KUKA KRL program: EPS_2_251806_MH58A_A_20260212042255.src

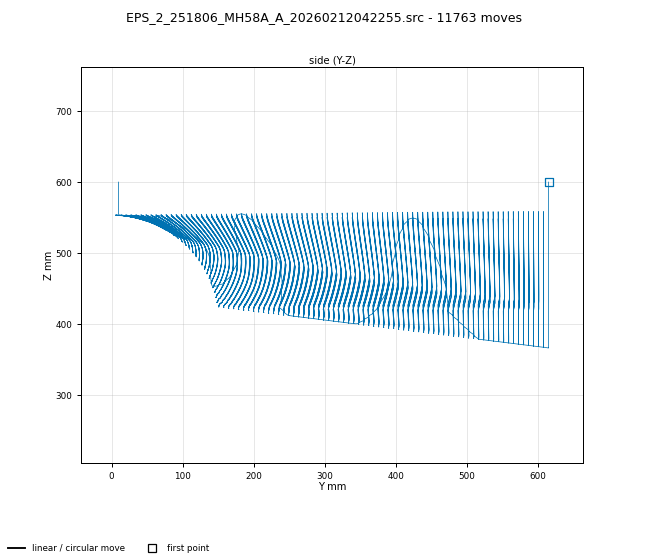
[picture p0: tool path of EPS_2_251806_MH58A_A_20260212042255.src, 11763 of 11765 moves have a stored position in this frame; points joined in program order, loops and branches not executed]
&ACCESS RVP
&REL 4
&COMMENT QRS 19112012
&PARAM EDITMASK = *
DEF PART()
EXT BAS (BAS_COMMAND :IN,REAL :IN )
INT I
BAS (#INITMOV,0 )

;KUKA QRS Post kuka4.cps  Date:22-06-2017 !

File_ID=3025

QRS_PRE_INIT()

;Init var - Until changes are made in qrs_pre_init
Outlet_Square_prg=0
Inlet_1_Square_prg=0
Inlet_2_Square_prg=0
Inlet_3_Square_prg=0
Inlet_4_Square_prg=0
Inlet_5_Square_prg=0

Outlet_1={X 0.000, Y 515.060, Z 433.000, B 0.000, E1 0.000 }
Inlet_1={X 0.000, Y 515.800, Z 423.000, B 0.000, E1 180.000 }
Outlet_1_type=251
Inlet_1_type=251
;QRS#1=Sidecore dimensions
;QRS#2=250-10" PVC SDR 35
;QRS#3=250-10" PVC SDR 35
;QRS#4=
;QRS#5=
;QRS#6=
;QRS#7=
;QRS#8=
;QRS#9=14M PSX
;QRS#10=14M PSX
;QRS#11=
;QRS#12=
;QRS#13=
;QRS#14=
;QRS#15=
;QRS#16=1220x127x838 2,75'
;QRS#17=EPS Height
;QRS#18=558,5
;QRS#19=*
;QRS#20= UPDATED VERSION 22-06-2017
;QRS#21=*
Outlet_Square=0100
Inlet_1_Square=0100
Inlet_2_Square=0
Inlet_3_Square=0
Inlet_4_Square=0
Inlet_5_Square=0
Mill_Square=1
Outlet_Square_Prg=205
Inlet_1_Square_prg=205

QRS_INIT()

$ADVANCE=5

; T1
PTP {E1 173.605,E2 173.605}
PTP {X 0,Y 615.509,A -85,B 0,C 180,E1 173.605,E2 173.605,E3 0,E4 0,E5 0,E6 0}
QRS_SPEED_INIT()
LIN {X 0,Y 615.509,Z 600,A -85,B 0,C 180,E1 173.605,E2 173.605,E3 0,E4 0,E5 0,E6 0} C_VEL
LIN {X 0,Y 615.509,Z 376.499,A -85,B 0,C 180,E1 173.605,E2 173.605} C_VEL
LIN {X 0,Y 615.509,Z 368.324,A -85,B 0,C 180,E1 173.605,E2 173.605} C_VEL
LIN {X 0,Y 615.493,Z 366.324,A -85,B 0,C 180,E1 173.419,E2 173.419} C_VEL
LIN {X 0,Y 615.489,Z 366.315,A -85,B 0,C 180,E1 170.801,E2 170.801} C_VEL
LIN {X 0,Y 615.48,Z 366.318,A -85,B 0,C 180,E1 168.139,E2 168.139} C_VEL
LIN {X 0,Y 615.484,Z 366.327,A -85,B 0,C 180,E1 165.451,E2 165.451} C_VEL
LIN {X 0,Y 615.495,Z 366.313,A -85,B 0,C 180,E1 162.73,E2 162.73} C_VEL
LIN {X 0,Y 615.49,Z 366.315,A -85,B 0,C 180,E1 159.967,E2 159.967} C_VEL
LIN {X 0,Y 615.497,Z 366.322,A -85,B 0,C 180,E1 157.156,E2 157.156} C_VEL
LIN {X 0,Y 615.481,Z 366.322,A -85,B 0,C 180,E1 154.284,E2 154.284} C_VEL
LIN {X 0,Y 615.478,Z 366.316,A -85,B 0,C 180,E1 151.552,E2 151.552} C_VEL
LIN {X 0,Y 615.487,Z 366.321,A -85,B 0,C 180,E1 148.914,E2 148.914} C_VEL
LIN {X 0,Y 615.478,Z 366.318,A -85,B 0,C 180,E1 146.467,E2 146.467} C_VEL
LIN {X 0,Y 615.497,Z 366.322,A -85,B 0,C 180,E1 144.165,E2 144.165} C_VEL
LIN {X 0,Y 615.483,Z 366.315,A -85,B 0,C 180,E1 141.931,E2 141.931} C_VEL
LIN {X 0,Y 615.49,Z 366.326,A -85,B 0,C 180,E1 139.394,E2 139.394} C_VEL
LIN {X 0,Y 615.478,Z 366.317,A -85,B 0,C 180,E1 136.754,E2 136.754} C_VEL
LIN {X 0,Y 615.481,Z 366.317,A -85,B 0,C 180,E1 133.997,E2 133.997} C_VEL
LIN {X 0,Y 615.488,Z 366.323,A -85,B 0,C 180,E1 131.474,E2 131.474} C_VEL
LIN {X 0,Y 615.478,Z 366.316,A -85,B 0,C 180,E1 128.905,E2 128.905} C_VEL
LIN {X 0,Y 615.486,Z 366.82,A -85,B 0,C 180,E1 128.011,E2 128.011} C_VEL
LIN {X 0,Y 615.487,Z 371.423,A -85,B 0,C 180,E1 125.616,E2 125.616} C_VEL
LIN {X 0,Y 615.485,Z 376.105,A -85,B 0,C 180,E1 123.236,E2 123.236} C_VEL
LIN {X 0,Y 615.478,Z 380.808,A -85,B 0,C 180,E1 120.92,E2 120.92} C_VEL
LIN {X 0,Y 615.491,Z 385.941,A -85,B 0,C 180,E1 118.45,E2 118.45} C_VEL
LIN {X 0,Y 615.498,Z 392.089,A -85,B 0,C 180,E1 115.57,E2 115.57} C_VEL
LIN {X 0,Y 615.492,Z 398.04,A -85,B 0,C 180,E1 112.844,E2 112.844} C_VEL
LIN {X 0,Y 615.479,Z 404.312,A -85,B 0,C 180,E1 110.033,E2 110.033} C_VEL
LIN {X 0,Y 615.481,Z 410.569,A -85,B 0,C 180,E1 107.271,E2 107.271} C_VEL
LIN {X 0,Y 615.481,Z 416.835,A -85,B 0,C 180,E1 104.549,E2 104.549} C_VEL
LIN {X 0,Y 615.483,Z 418.133,A -85,B 0,C 180,E1 103.989,E2 103.989} C_VEL
LIN {X 0,Y 615.486,Z 434.986,A -85,B 0,C 180,E1 103.664,E2 103.664} C_VEL
LIN {X 0,Y 615.478,Z 449.325,A -85,B 0,C 180,E1 103.243,E2 103.243} C_VEL
LIN {X 0,Y 615.487,Z 462.901,A -85,B 0,C 180,E1 102.698,E2 102.698} C_VEL
LIN {X 0,Y 615.486,Z 475.843,A -85,B 0,C 180,E1 102.028,E2 102.028} C_VEL
LIN {X 0,Y 615.499,Z 487.559,A -85,B 0,C 180,E1 101.276,E2 101.276} C_VEL
LIN {X 0,Y 615.498,Z 499.226,A -85,B 0,C 180,E1 100.36,E2 100.36} C_VEL
LIN {X 0,Y 615.497,Z 509.65,A -85,B 0,C 180,E1 99.364,E2 99.364} C_VEL
LIN {X 0,Y 615.496,Z 518.24,A -85,B 0,C 180,E1 98.371,E2 98.371} C_VEL
LIN {X 0,Y 615.495,Z 526.453,A -85,B 0,C 180,E1 97.216,E2 97.216} C_VEL
LIN {X 0,Y 615.496,Z 532.184,A -85,B 0,C 180,E1 96.227,E2 96.227} C_VEL
LIN {X 0,Y 615.494,Z 536.887,A -85,B 0,C 180,E1 95.241,E2 95.241} C_VEL
LIN {X 0,Y 615.496,Z 541.757,A -85,B 0,C 180,E1 93.928,E2 93.928} C_VEL
LIN {X 0,Y 615.496,Z 545.154,A -85,B 0,C 180,E1 92.618,E2 92.618} C_VEL
LIN {X 0,Y 615.493,Z 547.174,A -85,B 0,C 180,E1 91.309,E2 91.309} C_VEL
LIN {X 0,Y 615.494,Z 547.884,A -85,B 0,C 180,E1 90,E2 90} C_VEL
LIN {X 0,Y 615.49,Z 547.28,A -85,B 0,C 180,E1 88.691,E2 88.691} C_VEL
LIN {X 0,Y 615.493,Z 545.35,A -85,B 0,C 180,E1 87.382,E2 87.382} C_VEL
LIN {X 0,Y 615.496,Z 542.045,A -85,B 0,C 180,E1 86.071,E2 86.071} C_VEL
LIN {X 0,Y 615.496,Z 537.273,A -85,B 0,C 180,E1 84.759,E2 84.759} C_VEL
LIN {X 0,Y 615.495,Z 530.874,A -85,B 0,C 180,E1 83.443,E2 83.443} C_VEL
LIN {X 0,Y 615.496,Z 523.743,A -85,B 0,C 180,E1 82.289,E2 82.289} C_VEL
LIN {X 0,Y 615.497,Z 516.27,A -85,B 0,C 180,E1 81.298,E2 81.298} C_VEL
LIN {X 0,Y 615.496,Z 507.29,A -85,B 0,C 180,E1 80.304,E2 80.304} C_VEL
LIN {X 0,Y 615.499,Z 496.204,A -85,B 0,C 180,E1 79.291,E2 79.291} C_VEL
LIN {X 0,Y 615.498,Z 485.279,A -85,B 0,C 180,E1 78.473,E2 78.473} C_VEL
LIN {X 0,Y 615.479,Z 472.982,A -85,B 0,C 180,E1 77.721,E2 77.721} C_VEL
LIN {X 0,Y 615.488,Z 461.143,A -85,B 0,C 180,E1 77.134,E2 77.134} C_VEL
LIN {X 0,Y 615.476,Z 448.216,A -85,B 0,C 180,E1 76.63,E2 76.63} C_VEL
LIN {X 0,Y 615.492,Z 435.233,A -85,B 0,C 180,E1 76.252,E2 76.252} C_VEL
LIN {X 0,Y 615.482,Z 420.854,A -85,B 0,C 180,E1 75.971,E2 75.971} C_VEL
LIN {X 0,Y 615.48,Z 418.118,A -85,B 0,C 180,E1 75.914,E2 75.914} C_VEL
LIN {X 0,Y 615.489,Z 412.342,A -85,B 0,C 180,E1 73.413,E2 73.413} C_VEL
LIN {X 0,Y 615.484,Z 406.076,A -85,B 0,C 180,E1 70.662,E2 70.662} C_VEL
LIN {X 0,Y 615.478,Z 399.81,A -85,B 0,C 180,E1 67.863,E2 67.863} C_VEL
LIN {X 0,Y 615.492,Z 393.538,A -85,B 0,C 180,E1 65.008,E2 65.008} C_VEL
LIN {X 0,Y 615.484,Z 388.839,A -85,B 0,C 180,E1 62.823,E2 62.823} C_VEL
LIN {X 0,Y 615.482,Z 383.318,A -85,B 0,C 180,E1 60.207,E2 60.207} C_VEL
LIN {X 0,Y 615.489,Z 377.849,A -85,B 0,C 180,E1 57.542,E2 57.542} C_VEL
LIN {X 0,Y 615.483,Z 373.159,A -85,B 0,C 180,E1 55.184,E2 55.184} C_VEL
LIN {X 0,Y 615.488,Z 368.46,A -85,B 0,C 180,E1 52.758,E2 52.758} C_VEL
LIN {X 0,Y 615.494,Z 366.881,A -85,B 0,C 180,E1 51.932,E2 51.932} C_VEL
LIN {X 0,Y 615.482,Z 366.315,A -85,B 0,C 180,E1 50.939,E2 50.939} C_VEL
LIN {X 0,Y 615.493,Z 366.325,A -85,B 0,C 180,E1 48.526,E2 48.526} C_VEL
LIN {X 0,Y 615.491,Z 366.315,A -85,B 0,C 180,E1 45.85,E2 45.85} C_VEL
LIN {X 0,Y 615.483,Z 366.315,A -85,B 0,C 180,E1 43.047,E2 43.047} C_VEL
LIN {X 0,Y 615.495,Z 366.322,A -85,B 0,C 180,E1 40.606,E2 40.606} C_VEL
LIN {X 0,Y 615.483,Z 366.315,A -85,B 0,C 180,E1 38.011,E2 38.011} C_VEL
LIN {X 0,Y 615.498,Z 366.325,A -85,B 0,C 180,E1 35.615,E2 35.615} C_VEL
LIN {X 0,Y 615.482,Z 366.315,A -85,B 0,C 180,E1 33.237,E2 33.237} C_VEL
LIN {X 0,Y 615.494,Z 366.322,A -85,B 0,C 180,E1 30.919,E2 30.919} C_VEL
LIN {X 0,Y 615.478,Z 366.316,A -85,B 0,C 180,E1 28.448,E2 28.448} C_VEL
LIN {X 0,Y 615.489,Z 366.322,A -85,B 0,C 180,E1 25.716,E2 25.716} C_VEL
LIN {X 0,Y 615.495,Z 366.321,A -85,B 0,C 180,E1 22.844,E2 22.844} C_VEL
LIN {X 0,Y 615.491,Z 366.314,A -85,B 0,C 180,E1 20.033,E2 20.033} C_VEL
LIN {X 0,Y 615.494,Z 366.314,A -85,B 0,C 180,E1 17.27,E2 17.27} C_VEL
LIN {X 0,Y 615.489,Z 366.327,A -85,B 0,C 180,E1 14.549,E2 14.549} C_VEL
LIN {X 0,Y 615.477,Z 366.318,A -85,B 0,C 180,E1 11.861,E2 11.861} C_VEL
LIN {X 0,Y 615.489,Z 366.316,A -85,B 0,C 180,E1 9.199,E2 9.199} C_VEL
LIN {X 0,Y 615.492,Z 366.324,A -85,B 0,C 180,E1 6.557,E2 6.557} C_VEL
LIN {X 0,Y 615.478,Z 366.316,A -85,B 0,C 180,E1 3.929,E2 3.929} C_VEL
LIN {X 0,Y 615.487,Z 366.32,A -85,B 0,C 180,E1 1.309,E2 1.309} C_VEL
LIN {X 0,Y 615.487,Z 366.319,A -85,B 0,C 180,E1 -1.309,E2 -1.309} C_VEL
LIN {X 0,Y 615.477,Z 366.317,A -85,B 0,C 180,E1 -3.929,E2 -3.929} C_VEL
LIN {X 0,Y 615.493,Z 366.325,A -85,B 0,C 180,E1 -6.58,E2 -6.58} C_VEL
LIN {X 0,Y 615.489,Z 366.315,A -85,B 0,C 180,E1 -9.199,E2 -9.199} C_VEL
LIN {X 0,Y 615.48,Z 366.318,A -85,B 0,C 180,E1 -11.861,E2 -11.861} C_VEL
LIN {X 0,Y 615.491,Z 366.325,A -85,B 0,C 180,E1 -14.549,E2 -14.549} C_VEL
LIN {X 0,Y 615.492,Z 366.314,A -85,B 0,C 180,E1 -17.27,E2 -17.27} C_VEL
LIN {X 0,Y 615.493,Z 366.314,A -85,B 0,C 180,E1 -20.033,E2 -20.033} C_VEL
LIN {X 0,Y 615.495,Z 366.322,A -85,B 0,C 180,E1 -22.844,E2 -22.844} C_VEL
LIN {X 0,Y 615.478,Z 366.323,A -85,B 0,C 180,E1 -25.716,E2 -25.716} C_VEL
LIN {X 0,Y 615.478,Z 366.316,A -85,B 0,C 180,E1 -28.448,E2 -28.448} C_VEL
LIN {X 0,Y 615.486,Z 366.321,A -85,B 0,C 180,E1 -31.085,E2 -31.085} C_VEL
LIN {X 0,Y 615.478,Z 366.318,A -85,B 0,C 180,E1 -33.532,E2 -33.532} C_VEL
LIN {X 0,Y 615.496,Z 366.322,A -85,B 0,C 180,E1 -35.834,E2 -35.834} C_VEL
LIN {X 0,Y 615.483,Z 366.315,A -85,B 0,C 180,E1 -38.069,E2 -38.069} C_VEL
LIN {X 0,Y 615.494,Z 366.325,A -85,B 0,C 180,E1 -40.606,E2 -40.606} C_VEL
LIN {X 0,Y 615.478,Z 366.318,A -85,B 0,C 180,E1 -43.246,E2 -43.246} C_VEL
LIN {X 0,Y 615.482,Z 366.316,A -85,B 0,C 180,E1 -46.003,E2 -46.003} C_VEL
LIN {X 0,Y 615.488,Z 366.324,A -85,B 0,C 180,E1 -48.526,E2 -48.526} C_VEL
LIN {X 0,Y 615.478,Z 366.316,A -85,B 0,C 180,E1 -51.095,E2 -51.095} C_VEL
LIN {X 0,Y 615.492,Z 366.45,A -85,B 0,C 180,E1 -51.724,E2 -51.724} C_VEL
LIN {X 0,Y 615.487,Z 372.465,A -85,B 0,C 180,E1 -54.384,E2 -54.384} C_VEL
LIN {X 0,Y 615.485,Z 378.035,A -85,B 0,C 180,E1 -56.763,E2 -56.763} C_VEL
LIN {X 0,Y 615.478,Z 383.591,A -85,B 0,C 180,E1 -59.08,E2 -59.08} C_VEL
LIN {X 0,Y 615.491,Z 389.648,A -85,B 0,C 180,E1 -61.549,E2 -61.549} C_VEL
LIN {X 0,Y 615.498,Z 396.905,A -85,B 0,C 180,E1 -64.429,E2 -64.429} C_VEL
LIN {X 0,Y 615.493,Z 403.92,A -85,B 0,C 180,E1 -67.156,E2 -67.156} C_VEL
LIN {X 0,Y 615.479,Z 411.32,A -85,B 0,C 180,E1 -69.967,E2 -69.967} C_VEL
LIN {X 0,Y 615.487,Z 418.695,A -85,B 0,C 180,E1 -72.729,E2 -72.729} C_VEL
LIN {X 0,Y 615.483,Z 426.086,A -85,B 0,C 180,E1 -75.451,E2 -75.451} C_VEL
LIN {X 0,Y 615.485,Z 427.541,A -85,B 0,C 180,E1 -75.97,E2 -75.97} C_VEL
LIN {X 0,Y 615.494,Z 441.452,A -85,B 0,C 180,E1 -76.21,E2 -76.21} C_VEL
LIN {X 0,Y 615.479,Z 455.537,A -85,B 0,C 180,E1 -76.588,E2 -76.588} C_VEL
LIN {X 0,Y 615.488,Z 468.121,A -85,B 0,C 180,E1 -77.051,E2 -77.051} C_VEL
LIN {X 0,Y 615.484,Z 480.577,A -85,B 0,C 180,E1 -77.637,E2 -77.637} C_VEL
LIN {X 0,Y 615.498,Z 493.318,A -85,B 0,C 180,E1 -78.39,E2 -78.39} C_VEL
LIN {X 0,Y 615.498,Z 504.479,A -85,B 0,C 180,E1 -79.199,E2 -79.199} C_VEL
LIN {X 0,Y 615.499,Z 515.176,A -85,B 0,C 180,E1 -80.138,E2 -80.138} C_VEL
LIN {X 0,Y 615.498,Z 524.542,A -85,B 0,C 180,E1 -81.133,E2 -81.133} C_VEL
LIN {X 0,Y 615.494,Z 532.302,A -85,B 0,C 180,E1 -82.124,E2 -82.124} C_VEL
LIN {X 0,Y 615.496,Z 538.651,A -85,B 0,C 180,E1 -83.1,E2 -83.1} C_VEL
LIN {X 0,Y 615.499,Z 544.069,A -85,B 0,C 180,E1 -84.101,E2 -84.101} C_VEL
LIN {X 0,Y 615.495,Z 549.682,A -85,B 0,C 180,E1 -85.415,E2 -85.415} C_VEL
LIN {X 0,Y 615.495,Z 553.754,A -85,B 0,C 180,E1 -86.727,E2 -86.727} C_VEL
LIN {X 0,Y 615.499,Z 556.405,A -85,B 0,C 180,E1 -88.037,E2 -88.037} C_VEL
LIN {X 0,Y 615.494,Z 557.723,A -85,B 0,C 180,E1 -89.346,E2 -89.346} C_VEL
LIN {X 0,Y 615.494,Z 557.723,A -85,B 0,C 180,E1 -90.654,E2 -90.654} C_VEL
LIN {X 0,Y 615.499,Z 556.405,A -85,B 0,C 180,E1 -91.963,E2 -91.963} C_VEL
LIN {X 0,Y 615.495,Z 553.754,A -85,B 0,C 180,E1 -93.273,E2 -93.273} C_VEL
LIN {X 0,Y 615.495,Z 549.683,A -85,B 0,C 180,E1 -94.584,E2 -94.584} C_VEL
LIN {X 0,Y 615.499,Z 544.07,A -85,B 0,C 180,E1 -95.898,E2 -95.898} C_VEL
LIN {X 0,Y 615.496,Z 538.652,A -85,B 0,C 180,E1 -96.9,E2 -96.9} C_VEL
LIN {X 0,Y 615.496,Z 531.073,A -85,B 0,C 180,E1 -98.041,E2 -98.041} C_VEL
LIN {X 0,Y 615.498,Z 521.588,A -85,B 0,C 180,E1 -99.199,E2 -99.199} C_VEL
LIN {X 0,Y 615.498,Z 511.642,A -85,B 0,C 180,E1 -100.194,E2 -100.194} C_VEL
LIN {X 0,Y 615.498,Z 500.384,A -85,B 0,C 180,E1 -101.118,E2 -101.118} C_VEL
LIN {X 0,Y 615.497,Z 489.415,A -85,B 0,C 180,E1 -101.861,E2 -101.861} C_VEL
LIN {X 0,Y 615.486,Z 477.329,A -85,B 0,C 180,E1 -102.53,E2 -102.53} C_VEL
LIN {X 0,Y 615.48,Z 463.93,A -85,B 0,C 180,E1 -103.117,E2 -103.117} C_VEL
LIN {X 0,Y 615.485,Z 449.896,A -85,B 0,C 180,E1 -103.58,E2 -103.58} C_VEL
LIN {X 0,Y 615.493,Z 435.698,A -85,B 0,C 180,E1 -103.904,E2 -103.904} C_VEL
LIN {X 0,Y 615.484,Z 427.449,A -85,B 0,C 180,E1 -104.049,E2 -104.049} C_VEL
LIN {X 0,Y 615.489,Z 420.545,A -85,B 0,C 180,E1 -106.587,E2 -106.587} C_VEL
LIN {X 0,Y 615.487,Z 413.158,A -85,B 0,C 180,E1 -109.338,E2 -109.338} C_VEL
LIN {X 0,Y 615.478,Z 405.775,A -85,B 0,C 180,E1 -112.137,E2 -112.137} C_VEL
LIN {X 0,Y 615.49,Z 398.379,A -85,B 0,C 180,E1 -114.992,E2 -114.992} C_VEL
LIN {X 0,Y 615.481,Z 392.839,A -85,B 0,C 180,E1 -117.177,E2 -117.177} C_VEL
LIN {X 0,Y 615.477,Z 386.338,A -85,B 0,C 180,E1 -119.793,E2 -119.793} C_VEL
LIN {X 0,Y 615.495,Z 379.886,A -85,B 0,C 180,E1 -122.457,E2 -122.457} C_VEL
LIN {X 0,Y 615.484,Z 374.318,A -85,B 0,C 180,E1 -124.815,E2 -124.815} C_VEL
LIN {X 0,Y 615.486,Z 368.759,A -85,B 0,C 180,E1 -127.242,E2 -127.242} C_VEL
LIN {X 0,Y 615.487,Z 366.32,A -85,B 0,C 180,E1 -128.381,E2 -128.381} C_VEL
LIN {X 0,Y 615.484,Z 366.321,A -85,B 0,C 180,E1 -131.094,E2 -131.094} C_VEL
LIN {X 0,Y 615.492,Z 366.319,A -85,B 0,C 180,E1 -133.244,E2 -133.244} C_VEL
LIN {X 0,Y 615.483,Z 366.323,A -85,B 0,C 180,E1 -136.003,E2 -136.003} C_VEL
LIN {X 0,Y 615.482,Z 366.317,A -85,B 0,C 180,E1 -138.906,E2 -138.906} C_VEL
LIN {X 0,Y 615.495,Z 366.326,A -85,B 0,C 180,E1 -141.096,E2 -141.096} C_VEL
LIN {X 0,Y 615.478,Z 366.316,A -85,B 0,C 180,E1 -143.575,E2 -143.575} C_VEL
LIN {X 0,Y 615.495,Z 366.325,A -85,B 0,C 180,E1 -145.978,E2 -145.978} C_VEL
LIN {X 0,Y 615.482,Z 366.315,A -85,B 0,C 180,E1 -148.314,E2 -148.314} C_VEL
LIN {X 0,Y 615.486,Z 366.322,A -85,B 0,C 180,E1 -150.594,E2 -150.594} C_VEL
LIN {X 0,Y 615.497,Z 366.314,A -85,B 0,C 180,E1 -152.953,E2 -152.953} C_VEL
LIN {X 0,Y 615.491,Z 366.319,A -85,B 0,C 180,E1 -155.991,E2 -155.991} C_VEL
LIN {X 0,Y 615.48,Z 366.32,A -85,B 0,C 180,E1 -158.568,E2 -158.568} C_VEL
LIN {X 0,Y 615.477,Z 366.316,A -85,B 0,C 180,E1 -161.354,E2 -161.354} C_VEL
LIN {X 0,Y 615.481,Z 366.321,A -85,B 0,C 180,E1 -164.095,E2 -164.095} C_VEL
LIN {X 0,Y 615.495,Z 366.319,A -85,B 0,C 180,E1 -166.799,E2 -166.799} C_VEL
LIN {X 0,Y 615.486,Z 366.314,A -85,B 0,C 180,E1 -169.473,E2 -169.473} C_VEL
LIN {X 0,Y 615.484,Z 366.322,A -85,B 0,C 180,E1 -172.124,E2 -172.124} C_VEL
LIN {X 0,Y 615.488,Z 366.318,A -85,B 0,C 180,E1 -174.759,E2 -174.759} C_VEL
LIN {X 0,Y 615.491,Z 366.314,A -85,B 0,C 180,E1 -177.382,E2 -177.382} C_VEL
LIN {X 0,Y 615.489,Z 366.327,A -85,B 0,C 180,E1 -180,E2 -180} C_VEL
LIN {X 0,Y 615.488,Z 366.314,A -85,B 0,C 180,E1 -182.618,E2 -182.618} C_VEL
LIN {X 0,Y 615.494,Z 366.317,A -85,B 0,C 180,E1 -185.241,E2 -185.241} C_VEL
LIN {X 0,Y 615.493,Z 366.324,A -85,B 0,C 180,E1 -186.581,E2 -186.581} C_VEL
LIN {X 0,Y 614.813,Z 366.462,A -85,B 0,C 180,E1 -187.127,E2 -187.127} C_VEL
LIN {X 0,Y 611.978,Z 366.882,A -85,B 0,C 180,E1 -188.013,E2 -188.013} C_VEL
LIN {X 0,Y 609.587,Z 367.19,A -85,B 0,C 180,E1 -188.726,E2 -188.726} C_VEL
LIN {X 0,Y 608.55,Z 367.306,A -85,B 0,C 180,E1 -189.275,E2 -189.275} C_VEL
LIN {X 0,Y 608.46,Z 367.316,A -85,B 0,C 180,E1 -189.461,E2 -189.461} C_VEL
LIN {X 0,Y 608.457,Z 367.316,A -85,B 0,C 180,E1 -192,E2 -192} C_VEL
LIN {X 0,Y 608.475,Z 367.319,A -85,B 0,C 180,E1 -194.721,E2 -194.721} C_VEL
LIN {X 0,Y 608.46,Z 367.317,A -85,B 0,C 180,E1 -197.476,E2 -197.476} C_VEL
LIN {X 0,Y 608.461,Z 367.315,A -85,B 0,C 180,E1 -200.274,E2 -200.274} C_VEL
LIN {X 0,Y 608.453,Z 367.318,A -85,B 0,C 180,E1 -203.124,E2 -203.124} C_VEL
LIN {X 0,Y 608.467,Z 367.318,A -85,B 0,C 180,E1 -205.72,E2 -205.72} C_VEL
LIN {X 0,Y 608.446,Z 367.317,A -85,B 0,C 180,E1 -208.267,E2 -208.267} C_VEL
LIN {X 0,Y 608.476,Z 367.316,A -85,B 0,C 180,E1 -210.545,E2 -210.545} C_VEL
LIN {X 0,Y 608.458,Z 367.317,A -85,B 0,C 180,E1 -212.88,E2 -212.88} C_VEL
LIN {X 0,Y 608.45,Z 367.318,A -85,B 0,C 180,E1 -215.277,E2 -215.277} C_VEL
LIN {X 0,Y 608.47,Z 367.315,A -85,B 0,C 180,E1 -217.746,E2 -217.746} C_VEL
LIN {X 0,Y 608.452,Z 367.32,A -85,B 0,C 180,E1 -220.329,E2 -220.329} C_VEL
LIN {X 0,Y 608.451,Z 367.316,A -85,B 0,C 180,E1 -222.96,E2 -222.96} C_VEL
LIN {X 0,Y 608.46,Z 367.318,A -85,B 0,C 180,E1 -225.736,E2 -225.736} C_VEL
LIN {X 0,Y 608.462,Z 367.322,A -85,B 0,C 180,E1 -228.658,E2 -228.658} C_VEL
LIN {X 0,Y 608.418,Z 367.322,A -85,B 0,C 180,E1 -231.408,E2 -231.408} C_VEL
LIN {X 0,Y 608.427,Z 367.488,A -85,B 0,C 180,E1 -231.765,E2 -231.765} C_VEL
LIN {X 0,Y 608.479,Z 371.628,A -85,B 0,C 180,E1 -233.951,E2 -233.951} C_VEL
LIN {X 0,Y 608.475,Z 376.254,A -85,B 0,C 180,E1 -236.33,E2 -236.33} C_VEL
LIN {X 0,Y 608.447,Z 381.065,A -85,B 0,C 180,E1 -238.733,E2 -238.733} C_VEL
LIN {X 0,Y 608.444,Z 386.537,A -85,B 0,C 180,E1 -241.385,E2 -241.385} C_VEL
LIN {X 0,Y 608.445,Z 391.99,A -85,B 0,C 180,E1 -243.964,E2 -243.964} C_VEL
LIN {X 0,Y 608.444,Z 396.717,A -85,B 0,C 180,E1 -246.154,E2 -246.154} C_VEL
LIN {X 0,Y 608.439,Z 403.019,A -85,B 0,C 180,E1 -249.018,E2 -249.018} C_VEL
LIN {X 0,Y 608.446,Z 409.321,A -85,B 0,C 180,E1 -251.828,E2 -251.828} C_VEL
LIN {X 0,Y 608.413,Z 415.624,A -85,B 0,C 180,E1 -254.593,E2 -254.593} C_VEL
LIN {X 0,Y 608.429,Z 418.531,A -85,B 0,C 180,E1 -255.856,E2 -255.856} C_VEL
LIN {X 0,Y 608.598,Z 434.098,A -85,B 0,C 180,E1 -256.157,E2 -256.157} C_VEL
LIN {X 0,Y 608.553,Z 448.066,A -85,B 0,C 180,E1 -256.561,E2 -256.561} C_VEL
LIN {X 0,Y 608.54,Z 461.051,A -85,B 0,C 180,E1 -257.07,E2 -257.07} C_VEL
LIN {X 0,Y 608.529,Z 472.942,A -85,B 0,C 180,E1 -257.663,E2 -257.663} C_VEL
LIN {X 0,Y 608.509,Z 485.299,A -85,B 0,C 180,E1 -258.424,E2 -258.424} C_VEL
LIN {X 0,Y 608.501,Z 497.474,A -85,B 0,C 180,E1 -259.351,E2 -259.351} C_VEL
LIN {X 0,Y 608.469,Z 508.272,A -85,B 0,C 180,E1 -260.359,E2 -260.359} C_VEL
LIN {X 0,Y 608.47,Z 517.192,A -85,B 0,C 180,E1 -261.364,E2 -261.364} C_VEL
LIN {X 0,Y 608.47,Z 525.737,A -85,B 0,C 180,E1 -262.534,E2 -262.534} C_VEL
LIN {X 0,Y 608.443,Z 533.325,A -85,B 0,C 180,E1 -263.831,E2 -263.831} C_VEL
LIN {X 0,Y 608.435,Z 538.788,A -85,B 0,C 180,E1 -265.03,E2 -265.03} C_VEL
LIN {X 0,Y 608.434,Z 542.298,A -85,B 0,C 180,E1 -266.026,E2 -266.026} C_VEL
LIN {X 0,Y 608.424,Z 545.734,A -85,B 0,C 180,E1 -267.352,E2 -267.352} C_VEL
LIN {X 0,Y 608.446,Z 547.777,A -85,B 0,C 180,E1 -268.676,E2 -268.676} C_VEL
LIN {X 0,Y 608.434,Z 548.495,A -85,B 0,C 180,E1 -270,E2 -270} C_VEL
LIN {X 0,Y 608.443,Z 547.882,A -85,B 0,C 180,E1 -271.324,E2 -271.324} C_VEL
LIN {X 0,Y 608.421,Z 545.928,A -85,B 0,C 180,E1 -272.648,E2 -272.648} C_VEL
LIN {X 0,Y 608.434,Z 542.584,A -85,B 0,C 180,E1 -273.974,E2 -273.974} C_VEL
LIN {X 0,Y 608.44,Z 537.76,A -85,B 0,C 180,E1 -275.302,E2 -275.302} C_VEL
LIN {X 0,Y 608.443,Z 531.472,A -85,B 0,C 180,E1 -276.601,E2 -276.601} C_VEL
LIN {X 0,Y 608.453,Z 524.099,A -85,B 0,C 180,E1 -277.8,E2 -277.8} C_VEL
LIN {X 0,Y 608.476,Z 516.562,A -85,B 0,C 180,E1 -278.803,E2 -278.803} C_VEL
LIN {X 0,Y 608.488,Z 507.517,A -85,B 0,C 180,E1 -279.809,E2 -279.809} C_VEL
LIN {X 0,Y 608.507,Z 496.723,A -85,B 0,C 180,E1 -280.804,E2 -280.804} C_VEL
LIN {X 0,Y 608.524,Z 485.381,A -85,B 0,C 180,E1 -281.661,E2 -281.661} C_VEL
LIN {X 0,Y 608.53,Z 473.037,A -85,B 0,C 180,E1 -282.422,E2 -282.422} C_VEL
LIN {X 0,Y 608.551,Z 461.167,A -85,B 0,C 180,E1 -283.015,E2 -283.015} C_VEL
LIN {X 0,Y 608.563,Z 448.214,A -85,B 0,C 180,E1 -283.524,E2 -283.524} C_VEL
LIN {X 0,Y 608.593,Z 434.006,A -85,B 0,C 180,E1 -283.935,E2 -283.935} C_VEL
LIN {X 0,Y 608.579,Z 419.504,A -85,B 0,C 180,E1 -284.21,E2 -284.21} C_VEL
LIN {X 0,Y 608.432,Z 418.495,A -85,B 0,C 180,E1 -284.249,E2 -284.249} C_VEL
LIN {X 0,Y 608.447,Z 412.677,A -85,B 0,C 180,E1 -286.784,E2 -286.784} C_VEL
LIN {X 0,Y 608.429,Z 406.371,A -85,B 0,C 180,E1 -289.571,E2 -289.571} C_VEL
LIN {X 0,Y 608.435,Z 400.065,A -85,B 0,C 180,E1 -292.407,E2 -292.407} C_VEL
LIN {X 0,Y 608.453,Z 395.336,A -85,B 0,C 180,E1 -294.571,E2 -294.571} C_VEL
LIN {X 0,Y 608.447,Z 389.029,A -85,B 0,C 180,E1 -297.518,E2 -297.518} C_VEL
LIN {X 0,Y 608.446,Z 383.913,A -85,B 0,C 180,E1 -299.968,E2 -299.968} C_VEL
LIN {X 0,Y 608.459,Z 378.001,A -85,B 0,C 180,E1 -302.88,E2 -302.88} C_VEL
LIN {X 0,Y 608.445,Z 373.298,A -85,B 0,C 180,E1 -305.278,E2 -305.278} C_VEL
LIN {X 0,Y 608.474,Z 368.565,A -85,B 0,C 180,E1 -307.746,E2 -307.746} C_VEL
LIN {X 0,Y 608.414,Z 367.323,A -85,B 0,C 180,E1 -308.592,E2 -308.592} C_VEL
LIN {X 0,Y 608.465,Z 367.321,A -85,B 0,C 180,E1 -311.342,E2 -311.342} C_VEL
LIN {X 0,Y 608.46,Z 367.317,A -85,B 0,C 180,E1 -314.264,E2 -314.264} C_VEL
LIN {X 0,Y 608.45,Z 367.316,A -85,B 0,C 180,E1 -317.04,E2 -317.04} C_VEL
LIN {X 0,Y 608.455,Z 367.32,A -85,B 0,C 180,E1 -319.697,E2 -319.697} C_VEL
LIN {X 0,Y 608.469,Z 367.315,A -85,B 0,C 180,E1 -322.254,E2 -322.254} C_VEL
LIN {X 0,Y 608.483,Z 367.312,A -85,B 0,C 180,E1 -325.09,E2 -325.09} C_VEL
LIN {X 0,Y 608.469,Z 367.317,A -85,B 0,C 180,E1 -327.906,E2 -327.906} C_VEL
LIN {X 0,Y 608.47,Z 367.314,A -85,B 0,C 180,E1 -330.22,E2 -330.22} C_VEL
LIN {X 0,Y 608.488,Z 367.314,A -85,B 0,C 180,E1 -332.791,E2 -332.791} C_VEL
LIN {X 0,Y 608.46,Z 367.318,A -85,B 0,C 180,E1 -335.429,E2 -335.429} C_VEL
LIN {X 0,Y 608.468,Z 367.314,A -85,B 0,C 180,E1 -338.308,E2 -338.308} C_VEL
LIN {X 0,Y 608.466,Z 367.314,A -85,B 0,C 180,E1 -341.286,E2 -341.286} C_VEL
LIN {X 0,Y 608.459,Z 367.321,A -85,B 0,C 180,E1 -343.906,E2 -343.906} C_VEL
LIN {X 0,Y 608.47,Z 367.315,A -85,B 0,C 180,E1 -346.644,E2 -346.644} C_VEL
LIN {X 0,Y 608.462,Z 367.315,A -85,B 0,C 180,E1 -349.35,E2 -349.35} C_VEL
LIN {X 0,Y 608.481,Z 367.318,A -85,B 0,C 180,E1 -352.033,E2 -352.033} C_VEL
LIN {X 0,Y 608.471,Z 367.315,A -85,B 0,C 180,E1 -354.698,E2 -354.698} C_VEL
LIN {X 0,Y 608.48,Z 367.313,A -85,B 0,C 180,E1 -357.352,E2 -357.352} C_VEL
LIN {X 0,Y 608.477,Z 367.32,A -85,B 0,C 180,E1 -360,E2 -360} C_VEL
LIN {X 0,Y 608.482,Z 367.313,A -85,B 0,C 180,E1 -362.648,E2 -362.648} C_VEL
LIN {X 0,Y 608.467,Z 367.316,A -85,B 0,C 180,E1 -365.302,E2 -365.302} C_VEL
LIN {X 0,Y 608.473,Z 367.318,A -85,B 0,C 180,E1 -367.967,E2 -367.967} C_VEL
LIN {X 0,Y 608.461,Z 367.315,A -85,B 0,C 180,E1 -370.65,E2 -370.65} C_VEL
LIN {X 0,Y 608.469,Z 367.316,A -85,B 0,C 180,E1 -373.356,E2 -373.356} C_VEL
LIN {X 0,Y 608.456,Z 367.321,A -85,B 0,C 180,E1 -376.094,E2 -376.094} C_VEL
LIN {X 0,Y 608.456,Z 367.316,A -85,B 0,C 180,E1 -378.87,E2 -378.87} C_VEL
LIN {X 0,Y 608.468,Z 367.315,A -85,B 0,C 180,E1 -381.692,E2 -381.692} C_VEL
LIN {X 0,Y 608.46,Z 367.319,A -85,B 0,C 180,E1 -384.571,E2 -384.571} C_VEL
LIN {X 0,Y 608.454,Z 367.322,A -85,B 0,C 180,E1 -387.518,E2 -387.518} C_VEL
LIN {X 0,Y 608.47,Z 367.314,A -85,B 0,C 180,E1 -389.972,E2 -389.972} C_VEL
LIN {X 0,Y 608.459,Z 367.317,A -85,B 0,C 180,E1 -392.879,E2 -392.879} C_VEL
LIN {X 0,Y 608.447,Z 367.318,A -85,B 0,C 180,E1 -395.277,E2 -395.277} C_VEL
LIN {X 0,Y 608.469,Z 367.316,A -85,B 0,C 180,E1 -397.746,E2 -397.746} C_VEL
LIN {X 0,Y 608.457,Z 367.319,A -85,B 0,C 180,E1 -400.329,E2 -400.329} C_VEL
LIN {X 0,Y 608.449,Z 367.316,A -85,B 0,C 180,E1 -402.96,E2 -402.96} C_VEL
LIN {X 0,Y 608.46,Z 367.318,A -85,B 0,C 180,E1 -405.736,E2 -405.736} C_VEL
LIN {X 0,Y 608.462,Z 367.322,A -85,B 0,C 180,E1 -408.658,E2 -408.658} C_VEL
LIN {X 0,Y 608.489,Z 367.405,A -85,B 0,C 180,E1 -411.617,E2 -411.617} C_VEL
LIN {X 0,Y 608.479,Z 372.612,A -85,B 0,C 180,E1 -413.95,E2 -413.95} C_VEL
LIN {X 0,Y 608.49,Z 378.114,A -85,B 0,C 180,E1 -416.331,E2 -416.331} C_VEL
LIN {X 0,Y 608.477,Z 383.804,A -85,B 0,C 180,E1 -418.728,E2 -418.728} C_VEL
LIN {X 0,Y 608.475,Z 390.252,A -85,B 0,C 180,E1 -421.38,E2 -421.38} C_VEL
LIN {X 0,Y 608.476,Z 397.488,A -85,B 0,C 180,E1 -424.279,E2 -424.279} C_VEL
LIN {X 0,Y 608.454,Z 404.127,A -85,B 0,C 180,E1 -426.876,E2 -426.876} C_VEL
LIN {X 0,Y 608.441,Z 411.556,A -85,B 0,C 180,E1 -429.725,E2 -429.725} C_VEL
LIN {X 0,Y 608.452,Z 418.984,A -85,B 0,C 180,E1 -432.523,E2 -432.523} C_VEL
LIN {X 0,Y 608.439,Z 426.413,A -85,B 0,C 180,E1 -435.278,E2 -435.278} C_VEL
LIN {X 0,Y 608.444,Z 427.83,A -85,B 0,C 180,E1 -435.8,E2 -435.8} C_VEL
LIN {X 0,Y 608.593,Z 443.894,A -85,B 0,C 180,E1 -436.107,E2 -436.107} C_VEL
LIN {X 0,Y 608.558,Z 458.139,A -85,B 0,C 180,E1 -436.518,E2 -436.518} C_VEL
LIN {X 0,Y 608.54,Z 472.09,A -85,B 0,C 180,E1 -437.07,E2 -437.07} C_VEL
LIN {X 0,Y 608.537,Z 485.266,A -85,B 0,C 180,E1 -437.748,E2 -437.748} C_VEL
LIN {X 0,Y 608.518,Z 497.147,A -85,B 0,C 180,E1 -438.508,E2 -438.508} C_VEL
LIN {X 0,Y 608.501,Z 507.99,A -85,B 0,C 180,E1 -439.351,E2 -439.351} C_VEL
LIN {X 0,Y 608.468,Z 518.707,A -85,B 0,C 180,E1 -440.359,E2 -440.359} C_VEL
LIN {X 0,Y 608.471,Z 527.556,A -85,B 0,C 180,E1 -441.364,E2 -441.364} C_VEL
LIN {X 0,Y 608.47,Z 536.038,A -85,B 0,C 180,E1 -442.534,E2 -442.534} C_VEL
LIN {X 0,Y 608.444,Z 543.545,A -85,B 0,C 180,E1 -443.831,E2 -443.831} C_VEL
LIN {X 0,Y 608.437,Z 548.961,A -85,B 0,C 180,E1 -445.03,E2 -445.03} C_VEL
LIN {X 0,Y 608.431,Z 552.441,A -85,B 0,C 180,E1 -446.026,E2 -446.026} C_VEL
LIN {X 0,Y 608.424,Z 555.831,A -85,B 0,C 180,E1 -447.352,E2 -447.352} C_VEL
LIN {X 0,Y 608.442,Z 557.83,A -85,B 0,C 180,E1 -448.676,E2 -448.676} C_VEL
LIN {X 0,Y 608.433,Z 558.5,A -85,B 0,C 180,E1 -450,E2 -450} C_VEL
LIN {X 0,Y 608.442,Z 557.83,A -85,B 0,C 180,E1 -451.324,E2 -451.324} C_VEL
LIN {X 0,Y 608.424,Z 555.831,A -85,B 0,C 180,E1 -452.648,E2 -452.648} C_VEL
LIN {X 0,Y 608.431,Z 552.441,A -85,B 0,C 180,E1 -453.974,E2 -453.974} C_VEL
LIN {X 0,Y 608.44,Z 547.568,A -85,B 0,C 180,E1 -455.302,E2 -455.302} C_VEL
LIN {X 0,Y 608.445,Z 541.211,A -85,B 0,C 180,E1 -456.603,E2 -456.603} C_VEL
LIN {X 0,Y 608.453,Z 533.798,A -85,B 0,C 180,E1 -457.8,E2 -457.8} C_VEL
LIN {X 0,Y 608.473,Z 524.823,A -85,B 0,C 180,E1 -458.971,E2 -458.971} C_VEL
LIN {X 0,Y 608.473,Z 515.391,A -85,B 0,C 180,E1 -459.977,E2 -459.977} C_VEL
LIN {X 0,Y 608.506,Z 504.046,A -85,B 0,C 180,E1 -460.973,E2 -460.973} C_VEL
LIN {X 0,Y 608.534,Z 492.148,A -85,B 0,C 180,E1 -461.829,E2 -461.829} C_VEL
LIN {X 0,Y 608.524,Z 479.072,A -85,B 0,C 180,E1 -462.591,E2 -462.591} C_VEL
LIN {X 0,Y 608.546,Z 466.172,A -85,B 0,C 180,E1 -463.185,E2 -463.185} C_VEL
LIN {X 0,Y 608.589,Z 452.18,A -85,B 0,C 180,E1 -463.673,E2 -463.673} C_VEL
LIN {X 0,Y 608.622,Z 438.451,A -85,B 0,C 180,E1 -464.013,E2 -464.013} C_VEL
LIN {X 0,Y 608.436,Z 427.852,A -85,B 0,C 180,E1 -464.192,E2 -464.192} C_VEL
LIN {X 0,Y 608.448,Z 420.842,A -85,B 0,C 180,E1 -466.784,E2 -466.784} C_VEL
LIN {X 0,Y 608.451,Z 413.413,A -85,B 0,C 180,E1 -469.571,E2 -469.571} C_VEL
LIN {X 0,Y 608.439,Z 407.842,A -85,B 0,C 180,E1 -471.693,E2 -471.693} C_VEL
LIN {X 0,Y 608.449,Z 401.5,A -85,B 0,C 180,E1 -474.146,E2 -474.146} C_VEL
LIN {X 0,Y 608.443,Z 394.842,A -85,B 0,C 180,E1 -476.775,E2 -476.775} C_VEL
LIN {X 0,Y 608.474,Z 389.27,A -85,B 0,C 180,E1 -479.02,E2 -479.02} C_VEL
LIN {X 0,Y 608.476,Z 383.699,A -85,B 0,C 180,E1 -481.316,E2 -481.316} C_VEL
LIN {X 0,Y 608.479,Z 377.96,A -85,B 0,C 180,E1 -483.736,E2 -483.736} C_VEL
LIN {X 0,Y 608.479,Z 372.52,A -85,B 0,C 180,E1 -486.09,E2 -486.09} C_VEL
LIN {X 0,Y 608.477,Z 367.316,A -85,B 0,C 180,E1 -488.486,E2 -488.486} C_VEL
LIN {X 0,Y 608.463,Z 367.322,A -85,B 0,C 180,E1 -491.342,E2 -491.342} C_VEL
LIN {X 0,Y 608.459,Z 367.318,A -85,B 0,C 180,E1 -494.264,E2 -494.264} C_VEL
LIN {X 0,Y 608.448,Z 367.316,A -85,B 0,C 180,E1 -497.04,E2 -497.04} C_VEL
LIN {X 0,Y 608.456,Z 367.319,A -85,B 0,C 180,E1 -499.697,E2 -499.697} C_VEL
LIN {X 0,Y 608.469,Z 367.315,A -85,B 0,C 180,E1 -502.254,E2 -502.254} C_VEL
LIN {X 0,Y 608.482,Z 367.312,A -85,B 0,C 180,E1 -505.09,E2 -505.09} C_VEL
LIN {X 0,Y 608.471,Z 367.316,A -85,B 0,C 180,E1 -507.906,E2 -507.906} C_VEL
LIN {X 0,Y 608.473,Z 367.314,A -85,B 0,C 180,E1 -510.221,E2 -510.221} C_VEL
LIN {X 0,Y 608.484,Z 367.314,A -85,B 0,C 180,E1 -512.792,E2 -512.792} C_VEL
LIN {X 0,Y 608.484,Z 367.317,A -85,B 0,C 180,E1 -515.846,E2 -515.846} C_VEL
LIN {X 0,Y 608.468,Z 367.314,A -85,B 0,C 180,E1 -518.308,E2 -518.308} C_VEL
LIN {X 0,Y 608.455,Z 367.316,A -85,B 0,C 180,E1 -521.13,E2 -521.13} C_VEL
LIN {X 0,Y 608.458,Z 367.321,A -85,B 0,C 180,E1 -523.906,E2 -523.906} C_VEL
LIN {X 0,Y 608.469,Z 367.316,A -85,B 0,C 180,E1 -526.644,E2 -526.644} C_VEL
LIN {X 0,Y 608.462,Z 367.315,A -85,B 0,C 180,E1 -529.35,E2 -529.35} C_VEL
LIN {X 0,Y 608.476,Z 367.318,A -85,B 0,C 180,E1 -532.033,E2 -532.033} C_VEL
LIN {X 0,Y 608.467,Z 367.316,A -85,B 0,C 180,E1 -534.698,E2 -534.698} C_VEL
LIN {X 0,Y 608.482,Z 367.313,A -85,B 0,C 180,E1 -537.352,E2 -537.352} C_VEL
LIN {X 0,Y 608.48,Z 367.32,A -85,B 0,C 180,E1 -540,E2 -540} C_VEL
LIN {X 0,Y 608.48,Z 367.313,A -85,B 0,C 180,E1 -542.648,E2 -542.648} C_VEL
LIN {X 0,Y 608.472,Z 367.315,A -85,B 0,C 180,E1 -545.302,E2 -545.302} C_VEL
LIN {X 0,Y 608.48,Z 367.317,A -85,B 0,C 180,E1 -547.967,E2 -547.967} C_VEL
LIN {X 0,Y 608.46,Z 367.316,A -85,B 0,C 180,E1 -549.461,E2 -549.461} C_VEL
LIN {X 0,Y 607.777,Z 367.404,A -85,B 0,C 180,E1 -550.014,E2 -550.014} C_VEL
LIN {X 0,Y 604.92,Z 367.757,A -85,B 0,C 180,E1 -550.911,E2 -550.911} C_VEL
LIN {X 0,Y 602.519,Z 368.059,A -85,B 0,C 180,E1 -551.632,E2 -551.632} C_VEL
LIN {X 0,Y 601.491,Z 368.183,A -85,B 0,C 180,E1 -552.189,E2 -552.189} C_VEL
LIN {X 0,Y 601.409,Z 368.194,A -85,B 0,C 180,E1 -552.377,E2 -552.377} C_VEL
LIN {X 0,Y 601.43,Z 368.194,A -85,B 0,C 180,E1 -554.897,E2 -554.897} C_VEL
LIN {X 0,Y 601.426,Z 368.191,A -85,B 0,C 180,E1 -556.986,E2 -556.986} C_VEL
LIN {X 0,Y 601.41,Z 368.196,A -85,B 0,C 180,E1 -559.809,E2 -559.809} C_VEL
LIN {X 0,Y 601.415,Z 368.199,A -85,B 0,C 180,E1 -562.683,E2 -562.683} C_VEL
LIN {X 0,Y 601.407,Z 368.194,A -85,B 0,C 180,E1 -564.878,E2 -564.878} C_VEL
LIN {X 0,Y 601.421,Z 368.195,A -85,B 0,C 180,E1 -567.867,E2 -567.867} C_VEL
LIN {X 0,Y 601.431,Z 368.191,A -85,B 0,C 180,E1 -570.164,E2 -570.164} C_VEL
LIN {X 0,Y 601.426,Z 368.195,A -85,B 0,C 180,E1 -572.716,E2 -572.716} C_VEL
LIN {X 0,Y 601.417,Z 368.193,A -85,B 0,C 180,E1 -575.115,E2 -575.115} C_VEL
LIN {X 0,Y 601.438,Z 368.196,A -85,B 0,C 180,E1 -577.419,E2 -577.419} C_VEL
LIN {X 0,Y 601.413,Z 368.193,A -85,B 0,C 180,E1 -579.995,E2 -579.995} C_VEL
LIN {X 0,Y 601.414,Z 368.194,A -85,B 0,C 180,E1 -582.67,E2 -582.67} C_VEL
LIN {X 0,Y 601.429,Z 368.198,A -85,B 0,C 180,E1 -585.482,E2 -585.482} C_VEL
LIN {X 0,Y 601.425,Z 368.195,A -85,B 0,C 180,E1 -588.407,E2 -588.407} C_VEL
LIN {X 0,Y 601.425,Z 368.193,A -85,B 0,C 180,E1 -590.875,E2 -590.875} C_VEL
LIN {X 0,Y 601.389,Z 368.421,A -85,B 0,C 180,E1 -591.73,E2 -591.73} C_VEL
LIN {X 0,Y 601.413,Z 373.14,A -85,B 0,C 180,E1 -594.247,E2 -594.247} C_VEL
LIN {X 0,Y 601.434,Z 377.834,A -85,B 0,C 180,E1 -596.687,E2 -596.687} C_VEL
LIN {X 0,Y 601.382,Z 382.54,A -85,B 0,C 180,E1 -599.056,E2 -599.056} C_VEL
LIN {X 0,Y 601.405,Z 387.266,A -85,B 0,C 180,E1 -601.372,E2 -601.372} C_VEL
LIN {X 0,Y 601.386,Z 393.054,A -85,B 0,C 180,E1 -604.138,E2 -604.138} C_VEL
LIN {X 0,Y 601.384,Z 398.293,A -85,B 0,C 180,E1 -606.588,E2 -606.588} C_VEL
LIN {X 0,Y 601.357,Z 404.596,A -85,B 0,C 180,E1 -609.476,E2 -609.476} C_VEL
LIN {X 0,Y 601.36,Z 410.898,A -85,B 0,C 180,E1 -612.311,E2 -612.311} C_VEL
LIN {X 0,Y 601.357,Z 417.201,A -85,B 0,C 180,E1 -615.101,E2 -615.101} C_VEL
LIN {X 0,Y 601.332,Z 418.544,A -85,B 0,C 180,E1 -615.691,E2 -615.691} C_VEL
LIN {X 0,Y 601.719,Z 421.869,A -85,B 0,C 180,E1 -615.749,E2 -615.749} C_VEL
LIN {X 0,Y 601.686,Z 435.955,A -85,B 0,C 180,E1 -616.038,E2 -616.038} C_VEL
LIN {X 0,Y 601.647,Z 448.63,A -85,B 0,C 180,E1 -616.422,E2 -616.422} C_VEL
LIN {X 0,Y 601.618,Z 461.065,A -85,B 0,C 180,E1 -616.919,E2 -616.919} C_VEL
LIN {X 0,Y 601.567,Z 472.954,A -85,B 0,C 180,E1 -617.518,E2 -617.518} C_VEL
LIN {X 0,Y 601.534,Z 485.308,A -85,B 0,C 180,E1 -618.288,E2 -618.288} C_VEL
LIN {X 0,Y 601.496,Z 496.305,A -85,B 0,C 180,E1 -619.124,E2 -619.124} C_VEL
LIN {X 0,Y 601.435,Z 506.651,A -85,B 0,C 180,E1 -620.075,E2 -620.075} C_VEL
LIN {X 0,Y 601.411,Z 515.837,A -85,B 0,C 180,E1 -621.093,E2 -621.093} C_VEL
LIN {X 0,Y 601.387,Z 524.62,A -85,B 0,C 180,E1 -622.277,E2 -622.277} C_VEL
LIN {X 0,Y 601.373,Z 531.382,A -85,B 0,C 180,E1 -623.395,E2 -623.395} C_VEL
LIN {X 0,Y 601.355,Z 537.378,A -85,B 0,C 180,E1 -624.635,E2 -624.635} C_VEL
LIN {X 0,Y 601.345,Z 542.3,A -85,B 0,C 180,E1 -625.979,E2 -625.979} C_VEL
LIN {X 0,Y 601.324,Z 545.735,A -85,B 0,C 180,E1 -627.32,E2 -627.32} C_VEL
LIN {X 0,Y 601.346,Z 547.779,A -85,B 0,C 180,E1 -628.661,E2 -628.661} C_VEL
LIN {X 0,Y 601.334,Z 548.496,A -85,B 0,C 180,E1 -630,E2 -630} C_VEL
LIN {X 0,Y 601.343,Z 547.882,A -85,B 0,C 180,E1 -631.339,E2 -631.339} C_VEL
LIN {X 0,Y 601.321,Z 545.927,A -85,B 0,C 180,E1 -632.68,E2 -632.68} C_VEL
LIN {X 0,Y 601.346,Z 542.583,A -85,B 0,C 180,E1 -634.021,E2 -634.021} C_VEL
LIN {X 0,Y 601.355,Z 537.758,A -85,B 0,C 180,E1 -635.365,E2 -635.365} C_VEL
LIN {X 0,Y 601.368,Z 531.887,A -85,B 0,C 180,E1 -636.601,E2 -636.601} C_VEL
LIN {X 0,Y 601.386,Z 525.216,A -85,B 0,C 180,E1 -637.724,E2 -637.724} C_VEL
LIN {X 0,Y 601.411,Z 516.558,A -85,B 0,C 180,E1 -638.907,E2 -638.907} C_VEL
LIN {X 0,Y 601.432,Z 507.511,A -85,B 0,C 180,E1 -639.925,E2 -639.925} C_VEL
LIN {X 0,Y 601.474,Z 496.335,A -85,B 0,C 180,E1 -640.964,E2 -640.964} C_VEL
LIN {X 0,Y 601.547,Z 484.097,A -85,B 0,C 180,E1 -641.883,E2 -641.883} C_VEL
LIN {X 0,Y 601.551,Z 471.463,A -85,B 0,C 180,E1 -642.654,E2 -642.654} C_VEL
LIN {X 0,Y 601.616,Z 459.187,A -85,B 0,C 180,E1 -643.253,E2 -643.253} C_VEL
LIN {X 0,Y 601.668,Z 446.218,A -85,B 0,C 180,E1 -643.748,E2 -643.748} C_VEL
LIN {X 0,Y 601.734,Z 432.448,A -85,B 0,C 180,E1 -644.133,E2 -644.133} C_VEL
LIN {X 0,Y 601.583,Z 420.132,A -85,B 0,C 180,E1 -644.369,E2 -644.369} C_VEL
LIN {X 0,Y 601.343,Z 418.538,A -85,B 0,C 180,E1 -644.402,E2 -644.402} C_VEL
LIN {X 0,Y 601.357,Z 412.676,A -85,B 0,C 180,E1 -646.988,E2 -646.988} C_VEL
LIN {X 0,Y 601.359,Z 406.37,A -85,B 0,C 180,E1 -649.811,E2 -649.811} C_VEL
LIN {X 0,Y 601.372,Z 400.064,A -85,B 0,C 180,E1 -652.685,E2 -652.685} C_VEL
LIN {X 0,Y 601.404,Z 393.758,A -85,B 0,C 180,E1 -655.619,E2 -655.619} C_VEL
LIN {X 0,Y 601.377,Z 389.028,A -85,B 0,C 180,E1 -657.87,E2 -657.87} C_VEL
LIN {X 0,Y 601.405,Z 384.298,A -85,B 0,C 180,E1 -660.165,E2 -660.165} C_VEL
LIN {X 0,Y 601.425,Z 379.188,A -85,B 0,C 180,E1 -662.715,E2 -662.715} C_VEL
LIN {X 0,Y 601.416,Z 374.537,A -85,B 0,C 180,E1 -665.114,E2 -665.114} C_VEL
LIN {X 0,Y 601.439,Z 370.155,A -85,B 0,C 180,E1 -667.419,E2 -667.419} C_VEL
LIN {X 0,Y 601.37,Z 368.231,A -85,B 0,C 180,E1 -668.463,E2 -668.463} C_VEL
LIN {X 0,Y 601.415,Z 368.194,A -85,B 0,C 180,E1 -670.875,E2 -670.875} C_VEL
LIN {X 0,Y 601.453,Z 368.189,A -85,B 0,C 180,E1 -673.584,E2 -673.584} C_VEL
LIN {X 0,Y 601.431,Z 368.196,A -85,B 0,C 180,E1 -676.427,E2 -676.427} C_VEL
LIN {X 0,Y 601.415,Z 368.195,A -85,B 0,C 180,E1 -679.125,E2 -679.125} C_VEL
LIN {X 0,Y 601.42,Z 368.192,A -85,B 0,C 180,E1 -681.732,E2 -681.732} C_VEL
LIN {X 0,Y 601.413,Z 368.198,A -85,B 0,C 180,E1 -684.247,E2 -684.247} C_VEL
LIN {X 0,Y 601.42,Z 368.192,A -85,B 0,C 180,E1 -686.686,E2 -686.686} C_VEL
LIN {X 0,Y 601.418,Z 368.197,A -85,B 0,C 180,E1 -689.058,E2 -689.058} C_VEL
LIN {X 0,Y 601.428,Z 368.192,A -85,B 0,C 180,E1 -691.373,E2 -691.373} C_VEL
LIN {X 0,Y 601.403,Z 368.195,A -85,B 0,C 180,E1 -693.636,E2 -693.636} C_VEL
LIN {X 0,Y 601.422,Z 368.192,A -85,B 0,C 180,E1 -696.59,E2 -696.59} C_VEL
LIN {X 0,Y 601.428,Z 368.192,A -85,B 0,C 180,E1 -699.478,E2 -699.478} C_VEL
LIN {X 0,Y 601.4,Z 368.2,A -85,B 0,C 180,E1 -702.312,E2 -702.312} C_VEL
LIN {X 0,Y 601.417,Z 368.193,A -85,B 0,C 180,E1 -704.409,E2 -704.409} C_VEL
LIN {X 0,Y 601.423,Z 368.197,A -85,B 0,C 180,E1 -707.172,E2 -707.172} C_VEL
LIN {X 0,Y 601.432,Z 368.192,A -85,B 0,C 180,E1 -709.905,E2 -709.905} C_VEL
LIN {X 0,Y 601.444,Z 368.189,A -85,B 0,C 180,E1 -712.615,E2 -712.615} C_VEL
LIN {X 0,Y 601.425,Z 368.196,A -85,B 0,C 180,E1 -715.308,E2 -715.308} C_VEL
LIN {X 0,Y 601.421,Z 368.194,A -85,B 0,C 180,E1 -717.991,E2 -717.991} C_VEL
LIN {X 0,Y 601.45,Z 368.188,A -85,B 0,C 180,E1 -720.669,E2 -720.669} C_VEL
LIN {X 0,Y 601.435,Z 368.196,A -85,B 0,C 180,E1 -723.349,E2 -723.349} C_VEL
LIN {X 0,Y 601.408,Z 368.195,A -85,B 0,C 180,E1 -726.037,E2 -726.037} C_VEL
LIN {X 0,Y 601.416,Z 368.193,A -85,B 0,C 180,E1 -728.738,E2 -728.738} C_VEL
LIN {X 0,Y 601.436,Z 368.196,A -85,B 0,C 180,E1 -731.458,E2 -731.458} C_VEL
LIN {X 0,Y 601.423,Z 368.193,A -85,B 0,C 180,E1 -734.205,E2 -734.205} C_VEL
LIN {X 0,Y 601.426,Z 368.191,A -85,B 0,C 180,E1 -736.986,E2 -736.986} C_VEL
LIN {X 0,Y 601.412,Z 368.196,A -85,B 0,C 180,E1 -739.809,E2 -739.809} C_VEL
LIN {X 0,Y 601.416,Z 368.199,A -85,B 0,C 180,E1 -742.683,E2 -742.683} C_VEL
LIN {X 0,Y 601.405,Z 368.195,A -85,B 0,C 180,E1 -744.878,E2 -744.878} C_VEL
LIN {X 0,Y 601.422,Z 368.195,A -85,B 0,C 180,E1 -747.867,E2 -747.867} C_VEL
LIN {X 0,Y 601.432,Z 368.191,A -85,B 0,C 180,E1 -750.164,E2 -750.164} C_VEL
LIN {X 0,Y 601.426,Z 368.195,A -85,B 0,C 180,E1 -752.716,E2 -752.716} C_VEL
LIN {X 0,Y 601.415,Z 368.193,A -85,B 0,C 180,E1 -755.114,E2 -755.114} C_VEL
LIN {X 0,Y 601.437,Z 368.196,A -85,B 0,C 180,E1 -757.419,E2 -757.419} C_VEL
LIN {X 0,Y 601.415,Z 368.194,A -85,B 0,C 180,E1 -759.995,E2 -759.995} C_VEL
LIN {X 0,Y 601.41,Z 368.195,A -85,B 0,C 180,E1 -762.67,E2 -762.67} C_VEL
LIN {X 0,Y 601.429,Z 368.197,A -85,B 0,C 180,E1 -765.482,E2 -765.482} C_VEL
LIN {X 0,Y 601.426,Z 368.195,A -85,B 0,C 180,E1 -768.407,E2 -768.407} C_VEL
LIN {X 0,Y 601.464,Z 368.239,A -85,B 0,C 180,E1 -771.478,E2 -771.478} C_VEL
LIN {X 0,Y 601.449,Z 374.36,A -85,B 0,C 180,E1 -774.249,E2 -774.249} C_VEL
LIN {X 0,Y 601.442,Z 379.968,A -85,B 0,C 180,E1 -776.687,E2 -776.687} C_VEL
LIN {X 0,Y 601.428,Z 385.556,A -85,B 0,C 180,E1 -779.058,E2 -779.058} C_VEL
LIN {X 0,Y 601.435,Z 391.127,A -85,B 0,C 180,E1 -781.373,E2 -781.373} C_VEL
LIN {X 0,Y 601.42,Z 398.556,A -85,B 0,C 180,E1 -784.382,E2 -784.382} C_VEL
LIN {X 0,Y 601.389,Z 406.202,A -85,B 0,C 180,E1 -787.401,E2 -787.401} C_VEL
LIN {X 0,Y 601.377,Z 413.413,A -85,B 0,C 180,E1 -790.189,E2 -790.189} C_VEL
LIN {X 0,Y 601.363,Z 420.842,A -85,B 0,C 180,E1 -793.012,E2 -793.012} C_VEL
LIN {X 0,Y 601.357,Z 427.853,A -85,B 0,C 180,E1 -795.638,E2 -795.638} C_VEL
LIN {X 0,Y 601.729,Z 432.291,A -85,B 0,C 180,E1 -795.711,E2 -795.711} C_VEL
LIN {X 0,Y 601.697,Z 446.727,A -85,B 0,C 180,E1 -796.013,E2 -796.013} C_VEL
LIN {X 0,Y 601.648,Z 459.923,A -85,B 0,C 180,E1 -796.421,E2 -796.421} C_VEL
LIN {X 0,Y 601.618,Z 472.091,A -85,B 0,C 180,E1 -796.918,E2 -796.918} C_VEL
LIN {X 0,Y 601.572,Z 485.264,A -85,B 0,C 180,E1 -797.604,E2 -797.604} C_VEL
LIN {X 0,Y 601.511,Z 497.148,A -85,B 0,C 180,E1 -798.372,E2 -798.372} C_VEL
LIN {X 0,Y 601.49,Z 507.991,A -85,B 0,C 180,E1 -799.225,E2 -799.225} C_VEL
LIN {X 0,Y 601.422,Z 518.707,A -85,B 0,C 180,E1 -800.245,E2 -800.245} C_VEL
LIN {X 0,Y 601.407,Z 527.557,A -85,B 0,C 180,E1 -801.262,E2 -801.262} C_VEL
LIN {X 0,Y 601.406,Z 536.039,A -85,B 0,C 180,E1 -802.446,E2 -802.446} C_VEL
LIN {X 0,Y 601.361,Z 542.75,A -85,B 0,C 180,E1 -803.604,E2 -803.604} C_VEL
LIN {X 0,Y 601.355,Z 547.567,A -85,B 0,C 180,E1 -804.635,E2 -804.635} C_VEL
LIN {X 0,Y 601.343,Z 552.441,A -85,B 0,C 180,E1 -805.979,E2 -805.979} C_VEL
LIN {X 0,Y 601.324,Z 555.831,A -85,B 0,C 180,E1 -807.32,E2 -807.32} C_VEL
LIN {X 0,Y 601.342,Z 557.831,A -85,B 0,C 180,E1 -808.661,E2 -808.661} C_VEL
LIN {X 0,Y 601.333,Z 558.5,A -85,B 0,C 180,E1 -810,E2 -810} C_VEL
LIN {X 0,Y 601.342,Z 557.831,A -85,B 0,C 180,E1 -811.339,E2 -811.339} C_VEL
LIN {X 0,Y 601.324,Z 555.832,A -85,B 0,C 180,E1 -812.68,E2 -812.68} C_VEL
LIN {X 0,Y 601.343,Z 552.442,A -85,B 0,C 180,E1 -814.021,E2 -814.021} C_VEL
LIN {X 0,Y 601.355,Z 547.568,A -85,B 0,C 180,E1 -815.365,E2 -815.365} C_VEL
LIN {X 0,Y 601.372,Z 541.622,A -85,B 0,C 180,E1 -816.605,E2 -816.605} C_VEL
LIN {X 0,Y 601.386,Z 534.919,A -85,B 0,C 180,E1 -817.723,E2 -817.723} C_VEL
LIN {X 0,Y 601.412,Z 526.198,A -85,B 0,C 180,E1 -818.907,E2 -818.907} C_VEL
LIN {X 0,Y 601.433,Z 517.082,A -85,B 0,C 180,E1 -819.925,E2 -819.925} C_VEL
LIN {X 0,Y 601.497,Z 506.828,A -85,B 0,C 180,E1 -820.877,E2 -820.877} C_VEL
LIN {X 0,Y 601.534,Z 495.971,A -85,B 0,C 180,E1 -821.712,E2 -821.712} C_VEL
LIN {X 0,Y 601.57,Z 483.776,A -85,B 0,C 180,E1 -822.482,E2 -822.482} C_VEL
LIN {X 0,Y 601.62,Z 470.127,A -85,B 0,C 180,E1 -823.167,E2 -823.167} C_VEL
LIN {X 0,Y 601.668,Z 456.901,A -85,B 0,C 180,E1 -823.68,E2 -823.68} C_VEL
LIN {X 0,Y 601.715,Z 442.653,A -85,B 0,C 180,E1 -824.084,E2 -824.084} C_VEL
LIN {X 0,Y 601.546,Z 429.189,A -85,B 0,C 180,E1 -824.338,E2 -824.338} C_VEL
LIN {X 0,Y 601.345,Z 427.853,A -85,B 0,C 180,E1 -824.363,E2 -824.363} C_VEL
LIN {X 0,Y 601.363,Z 420.842,A -85,B 0,C 180,E1 -826.988,E2 -826.988} C_VEL
LIN {X 0,Y 601.376,Z 413.413,A -85,B 0,C 180,E1 -829.81,E2 -829.81} C_VEL
LIN {X 0,Y 601.389,Z 406.202,A -85,B 0,C 180,E1 -832.599,E2 -832.599} C_VEL
LIN {X 0,Y 601.402,Z 400.413,A -85,B 0,C 180,E1 -834.879,E2 -834.879} C_VEL
LIN {X 0,Y 601.399,Z 394.236,A -85,B 0,C 180,E1 -837.359,E2 -837.359} C_VEL
LIN {X 0,Y 601.418,Z 389.27,A -85,B 0,C 180,E1 -839.393,E2 -839.393} C_VEL
LIN {X 0,Y 601.424,Z 383.693,A -85,B 0,C 180,E1 -841.726,E2 -841.726} C_VEL
LIN {X 0,Y 601.448,Z 378.09,A -85,B 0,C 180,E1 -844.117,E2 -844.117} C_VEL
LIN {X 0,Y 601.447,Z 372.505,A -85,B 0,C 180,E1 -846.58,E2 -846.58} C_VEL
LIN {X 0,Y 601.455,Z 368.192,A -85,B 0,C 180,E1 -848.589,E2 -848.589} C_VEL
LIN {X 0,Y 601.424,Z 368.194,A -85,B 0,C 180,E1 -851.765,E2 -851.765} C_VEL
LIN {X 0,Y 601.426,Z 368.198,A -85,B 0,C 180,E1 -854.535,E2 -854.535} C_VEL
LIN {X 0,Y 601.41,Z 368.195,A -85,B 0,C 180,E1 -857.41,E2 -857.41} C_VEL
LIN {X 0,Y 601.443,Z 368.19,A -85,B 0,C 180,E1 -860.464,E2 -860.464} C_VEL
LIN {X 0,Y 601.413,Z 368.193,A -85,B 0,C 180,E1 -863.418,E2 -863.418} C_VEL
LIN {X 0,Y 601.434,Z 368.196,A -85,B 0,C 180,E1 -866.064,E2 -866.064} C_VEL
LIN {X 0,Y 601.422,Z 368.192,A -85,B 0,C 180,E1 -868.545,E2 -868.545} C_VEL
LIN {X 0,Y 601.428,Z 368.192,A -85,B 0,C 180,E1 -871.373,E2 -871.373} C_VEL
LIN {X 0,Y 601.4,Z 368.196,A -85,B 0,C 180,E1 -873.636,E2 -873.636} C_VEL
LIN {X 0,Y 601.42,Z 368.192,A -85,B 0,C 180,E1 -876.59,E2 -876.59} C_VEL
LIN {X 0,Y 601.428,Z 368.192,A -85,B 0,C 180,E1 -879.478,E2 -879.478} C_VEL
LIN {X 0,Y 601.403,Z 368.199,A -85,B 0,C 180,E1 -882.312,E2 -882.312} C_VEL
LIN {X 0,Y 601.433,Z 368.193,A -85,B 0,C 180,E1 -885.103,E2 -885.103} C_VEL
LIN {X 0,Y 601.417,Z 368.192,A -85,B 0,C 180,E1 -887.858,E2 -887.858} C_VEL
LIN {X 0,Y 601.421,Z 368.195,A -85,B 0,C 180,E1 -890.584,E2 -890.584} C_VEL
LIN {X 0,Y 601.459,Z 368.191,A -85,B 0,C 180,E1 -893.324,E2 -893.324} C_VEL
LIN {X 0,Y 601.401,Z 368.194,A -85,B 0,C 180,E1 -895.979,E2 -895.979} C_VEL
LIN {X 0,Y 601.425,Z 368.195,A -85,B 0,C 180,E1 -898.661,E2 -898.661} C_VEL
LIN {X 0,Y 601.424,Z 368.194,A -85,B 0,C 180,E1 -901.339,E2 -901.339} C_VEL
LIN {X 0,Y 601.401,Z 368.194,A -85,B 0,C 180,E1 -904.021,E2 -904.021} C_VEL
LIN {X 0,Y 601.457,Z 368.191,A -85,B 0,C 180,E1 -906.71,E2 -906.71} C_VEL
LIN {X 0,Y 601.417,Z 368.195,A -85,B 0,C 180,E1 -909.459,E2 -909.459} C_VEL
LIN {X 0,Y 601.416,Z 368.192,A -85,B 0,C 180,E1 -912.143,E2 -912.143} C_VEL
LIN {X 0,Y 601.409,Z 368.194,A -85,B 0,C 180,E1 -912.377,E2 -912.377} C_VEL
LIN {X 0,Y 600.747,Z 368.282,A -85,B 0,C 180,E1 -912.937,E2 -912.937} C_VEL
LIN {X 0,Y 597.898,Z 368.634,A -85,B 0,C 180,E1 -913.845,E2 -913.845} C_VEL
LIN {X 0,Y 595.486,Z 368.938,A -85,B 0,C 180,E1 -914.575,E2 -914.575} C_VEL
LIN {X 0,Y 594.447,Z 369.062,A -85,B 0,C 180,E1 -915.139,E2 -915.139} C_VEL
LIN {X 0,Y 594.361,Z 369.071,A -85,B 0,C 180,E1 -915.329,E2 -915.329} C_VEL
LIN {X 0,Y 594.382,Z 369.075,A -85,B 0,C 180,E1 -917.904,E2 -917.904} C_VEL
LIN {X 0,Y 594.377,Z 369.074,A -85,B 0,C 180,E1 -920.915,E2 -920.915} C_VEL
LIN {X 0,Y 594.394,Z 369.068,A -85,B 0,C 180,E1 -923.704,E2 -923.704} C_VEL
LIN {X 0,Y 594.388,Z 369.068,A -85,B 0,C 180,E1 -926.7,E2 -926.7} C_VEL
LIN {X 0,Y 594.382,Z 369.073,A -85,B 0,C 180,E1 -928.999,E2 -928.999} C_VEL
LIN {X 0,Y 594.379,Z 369.069,A -85,B 0,C 180,E1 -931.643,E2 -931.643} C_VEL
LIN {X 0,Y 594.398,Z 369.068,A -85,B 0,C 180,E1 -934.579,E2 -934.579} C_VEL
LIN {X 0,Y 594.389,Z 369.072,A -85,B 0,C 180,E1 -937.087,E2 -937.087} C_VEL
LIN {X 0,Y 594.377,Z 369.069,A -85,B 0,C 180,E1 -939.774,E2 -939.774} C_VEL
LIN {X 0,Y 594.372,Z 369.075,A -85,B 0,C 180,E1 -942.375,E2 -942.375} C_VEL
LIN {X 0,Y 594.366,Z 369.074,A -85,B 0,C 180,E1 -945.191,E2 -945.191} C_VEL
LIN {X 0,Y 594.374,Z 369.071,A -85,B 0,C 180,E1 -947.625,E2 -947.625} C_VEL
LIN {X 0,Y 594.394,Z 369.074,A -85,B 0,C 180,E1 -950.321,E2 -950.321} C_VEL
LIN {X 0,Y 594.368,Z 369.073,A -85,B 0,C 180,E1 -951.298,E2 -951.298} C_VEL
LIN {X 0,Y 594.387,Z 370.626,A -85,B 0,C 180,E1 -952.392,E2 -952.392} C_VEL
LIN {X 0,Y 594.387,Z 374.877,A -85,B 0,C 180,E1 -954.672,E2 -954.672} C_VEL
LIN {X 0,Y 594.383,Z 379.507,A -85,B 0,C 180,E1 -957.088,E2 -957.088} C_VEL
LIN {X 0,Y 594.35,Z 384.602,A -85,B 0,C 180,E1 -959.678,E2 -959.678} C_VEL
LIN {X 0,Y 594.334,Z 390.418,A -85,B 0,C 180,E1 -962.537,E2 -962.537} C_VEL
LIN {X 0,Y 594.325,Z 395.144,A -85,B 0,C 180,E1 -964.805,E2 -964.805} C_VEL
LIN {X 0,Y 594.29,Z 401.446,A -85,B 0,C 180,E1 -967.764,E2 -967.764} C_VEL
LIN {X 0,Y 594.27,Z 406.173,A -85,B 0,C 180,E1 -969.943,E2 -969.943} C_VEL
LIN {X 0,Y 594.265,Z 410.899,A -85,B 0,C 180,E1 -972.092,E2 -972.092} C_VEL
LIN {X 0,Y 594.254,Z 415.626,A -85,B 0,C 180,E1 -974.216,E2 -974.216} C_VEL
LIN {X 0,Y 594.299,Z 418.679,A -85,B 0,C 180,E1 -975.521,E2 -975.521} C_VEL
LIN {X 0,Y 594.875,Z 424.213,A -85,B 0,C 180,E1 -975.621,E2 -975.621} C_VEL
LIN {X 0,Y 594.792,Z 438.297,A -85,B 0,C 180,E1 -975.937,E2 -975.937} C_VEL
LIN {X 0,Y 594.743,Z 452.795,A -85,B 0,C 180,E1 -976.417,E2 -976.417} C_VEL
LIN {X 0,Y 594.639,Z 466.479,A -85,B 0,C 180,E1 -977.023,E2 -977.023} C_VEL
LIN {X 0,Y 594.569,Z 478.774,A -85,B 0,C 180,E1 -977.716,E2 -977.716} C_VEL
LIN {X 0,Y 594.528,Z 491.046,A -85,B 0,C 180,E1 -978.569,E2 -978.569} C_VEL
LIN {X 0,Y 594.448,Z 501.36,A -85,B 0,C 180,E1 -979.441,E2 -979.441} C_VEL
LIN {X 0,Y 594.371,Z 511.46,A -85,B 0,C 180,E1 -980.471,E2 -980.471} C_VEL
LIN {X 0,Y 594.324,Z 519.845,A -85,B 0,C 180,E1 -981.5,E2 -981.5} C_VEL
LIN {X 0,Y 594.303,Z 527.859,A -85,B 0,C 180,E1 -982.697,E2 -982.697} C_VEL
LIN {X 0,Y 594.281,Z 534.313,A -85,B 0,C 180,E1 -983.89,E2 -983.89} C_VEL
LIN {X 0,Y 594.235,Z 540.036,A -85,B 0,C 180,E1 -985.251,E2 -985.251} C_VEL
LIN {X 0,Y 594.259,Z 544.199,A -85,B 0,C 180,E1 -986.61,E2 -986.61} C_VEL
LIN {X 0,Y 594.242,Z 546.927,A -85,B 0,C 180,E1 -987.967,E2 -987.967} C_VEL
LIN {X 0,Y 594.235,Z 548.302,A -85,B 0,C 180,E1 -989.322,E2 -989.322} C_VEL
LIN {X 0,Y 594.236,Z 548.356,A -85,B 0,C 180,E1 -990.678,E2 -990.678} C_VEL
LIN {X 0,Y 594.241,Z 547.073,A -85,B 0,C 180,E1 -992.033,E2 -992.033} C_VEL
LIN {X 0,Y 594.259,Z 544.432,A -85,B 0,C 180,E1 -993.39,E2 -993.39} C_VEL
LIN {X 0,Y 594.236,Z 540.362,A -85,B 0,C 180,E1 -994.749,E2 -994.749} C_VEL
LIN {X 0,Y 594.282,Z 534.74,A -85,B 0,C 180,E1 -996.11,E2 -996.11} C_VEL
LIN {X 0,Y 594.303,Z 528.391,A -85,B 0,C 180,E1 -997.304,E2 -997.304} C_VEL
LIN {X 0,Y 594.324,Z 520.494,A -85,B 0,C 180,E1 -998.5,E2 -998.5} C_VEL
LIN {X 0,Y 594.355,Z 512.239,A -85,B 0,C 180,E1 -999.529,E2 -999.529} C_VEL
LIN {X 0,Y 594.449,Z 502.301,A -85,B 0,C 180,E1 -1000.559,E2 -1000.559} C_VEL
LIN {X 0,Y 594.493,Z 491.162,A -85,B 0,C 180,E1 -1001.513,E2 -1001.513} C_VEL
LIN {X 0,Y 594.578,Z 478.826,A -85,B 0,C 180,E1 -1002.371,E2 -1002.371} C_VEL
LIN {X 0,Y 594.644,Z 466.538,A -85,B 0,C 180,E1 -1003.064,E2 -1003.064} C_VEL
LIN {X 0,Y 594.705,Z 452.869,A -85,B 0,C 180,E1 -1003.671,E2 -1003.671} C_VEL
LIN {X 0,Y 594.79,Z 438.921,A -85,B 0,C 180,E1 -1004.135,E2 -1004.135} C_VEL
LIN {X 0,Y 594.861,Z 424.697,A -85,B 0,C 180,E1 -1004.46,E2 -1004.46} C_VEL
LIN {X 0,Y 594.638,Z 420.516,A -85,B 0,C 180,E1 -1004.534,E2 -1004.534} C_VEL
LIN {X 0,Y 594.299,Z 418.499,A -85,B 0,C 180,E1 -1004.593,E2 -1004.593} C_VEL
LIN {X 0,Y 594.29,Z 412.675,A -85,B 0,C 180,E1 -1007.196,E2 -1007.196} C_VEL
LIN {X 0,Y 594.283,Z 407.945,A -85,B 0,C 180,E1 -1009.337,E2 -1009.337} C_VEL
LIN {X 0,Y 594.287,Z 403.216,A -85,B 0,C 180,E1 -1011.506,E2 -1011.506} C_VEL
LIN {X 0,Y 594.333,Z 396.967,A -85,B 0,C 180,E1 -1014.421,E2 -1014.421} C_VEL
LIN {X 0,Y 594.301,Z 392.18,A -85,B 0,C 180,E1 -1016.704,E2 -1016.704} C_VEL
LIN {X 0,Y 594.343,Z 387.45,A -85,B 0,C 180,E1 -1019.001,E2 -1019.001} C_VEL
LIN {X 0,Y 594.373,Z 382.164,A -85,B 0,C 180,E1 -1021.642,E2 -1021.642} C_VEL
LIN {X 0,Y 594.395,Z 376.477,A -85,B 0,C 180,E1 -1024.579,E2 -1024.579} C_VEL
LIN {X 0,Y 594.39,Z 371.746,A -85,B 0,C 180,E1 -1027.087,E2 -1027.087} C_VEL
LIN {X 0,Y 594.358,Z 369.075,A -85,B 0,C 180,E1 -1028.701,E2 -1028.701} C_VEL
LIN {X 0,Y 594.383,Z 369.075,A -85,B 0,C 180,E1 -1031.464,E2 -1031.464} C_VEL
LIN {X 0,Y 594.386,Z 369.07,A -85,B 0,C 180,E1 -1034.236,E2 -1034.236} C_VEL
LIN {X 0,Y 594.364,Z 369.071,A -85,B 0,C 180,E1 -1037.148,E2 -1037.148} C_VEL
LIN {X 0,Y 594.372,Z 369.076,A -85,B 0,C 180,E1 -1039.433,E2 -1039.433} C_VEL
LIN {X 0,Y 594.393,Z 369.07,A -85,B 0,C 180,E1 -1042.392,E2 -1042.392} C_VEL
LIN {X 0,Y 594.389,Z 369.071,A -85,B 0,C 180,E1 -1044.672,E2 -1044.672} C_VEL
LIN {X 0,Y 594.382,Z 369.07,A -85,B 0,C 180,E1 -1047.088,E2 -1047.088} C_VEL
LIN {X 0,Y 594.389,Z 369.069,A -85,B 0,C 180,E1 -1049.672,E2 -1049.672} C_VEL
LIN {X 0,Y 594.378,Z 369.076,A -85,B 0,C 180,E1 -1052.539,E2 -1052.539} C_VEL
LIN {X 0,Y 594.38,Z 369.069,A -85,B 0,C 180,E1 -1054.807,E2 -1054.807} C_VEL
LIN {X 0,Y 594.368,Z 369.076,A -85,B 0,C 180,E1 -1057.265,E2 -1057.265} C_VEL
LIN {X 0,Y 594.377,Z 369.069,A -85,B 0,C 180,E1 -1059.946,E2 -1059.946} C_VEL
LIN {X 0,Y 594.388,Z 369.068,A -85,B 0,C 180,E1 -1062.806,E2 -1062.806} C_VEL
LIN {X 0,Y 594.392,Z 369.069,A -85,B 0,C 180,E1 -1065.826,E2 -1065.826} C_VEL
LIN {X 0,Y 594.395,Z 369.07,A -85,B 0,C 180,E1 -1068.404,E2 -1068.404} C_VEL
LIN {X 0,Y 594.382,Z 369.069,A -85,B 0,C 180,E1 -1071.158,E2 -1071.158} C_VEL
LIN {X 0,Y 594.366,Z 369.073,A -85,B 0,C 180,E1 -1073.891,E2 -1073.891} C_VEL
LIN {X 0,Y 594.386,Z 369.072,A -85,B 0,C 180,E1 -1076.611,E2 -1076.611} C_VEL
LIN {X 0,Y 594.421,Z 369.064,A -85,B 0,C 180,E1 -1079.323,E2 -1079.323} C_VEL
LIN {X 0,Y 594.397,Z 369.069,A -85,B 0,C 180,E1 -1082.033,E2 -1082.033} C_VEL
LIN {X 0,Y 594.399,Z 369.072,A -85,B 0,C 180,E1 -1084.748,E2 -1084.748} C_VEL
LIN {X 0,Y 594.395,Z 369.067,A -85,B 0,C 180,E1 -1087.473,E2 -1087.473} C_VEL
LIN {X 0,Y 594.397,Z 369.068,A -85,B 0,C 180,E1 -1090.216,E2 -1090.216} C_VEL
LIN {X 0,Y 594.372,Z 369.077,A -85,B 0,C 180,E1 -1092.983,E2 -1092.983} C_VEL
LIN {X 0,Y 594.375,Z 369.071,A -85,B 0,C 180,E1 -1095.078,E2 -1095.078} C_VEL
LIN {X 0,Y 594.389,Z 369.068,A -85,B 0,C 180,E1 -1097.193,E2 -1097.193} C_VEL
LIN {X 0,Y 594.379,Z 369.07,A -85,B 0,C 180,E1 -1100.054,E2 -1100.054} C_VEL
LIN {X 0,Y 594.368,Z 369.074,A -85,B 0,C 180,E1 -1102.967,E2 -1102.967} C_VEL
LIN {X 0,Y 594.375,Z 369.069,A -85,B 0,C 180,E1 -1105.193,E2 -1105.193} C_VEL
LIN {X 0,Y 594.389,Z 369.074,A -85,B 0,C 180,E1 -1107.527,E2 -1107.527} C_VEL
LIN {X 0,Y 594.389,Z 369.069,A -85,B 0,C 180,E1 -1110.328,E2 -1110.328} C_VEL
LIN {X 0,Y 594.381,Z 369.07,A -85,B 0,C 180,E1 -1112.95,E2 -1112.95} C_VEL
LIN {X 0,Y 594.385,Z 369.072,A -85,B 0,C 180,E1 -1115.407,E2 -1115.407} C_VEL
LIN {X 0,Y 594.388,Z 369.069,A -85,B 0,C 180,E1 -1117.941,E2 -1117.941} C_VEL
LIN {X 0,Y 594.379,Z 369.073,A -85,B 0,C 180,E1 -1120.822,E2 -1120.822} C_VEL
LIN {X 0,Y 594.368,Z 369.072,A -85,B 0,C 180,E1 -1123.299,E2 -1123.299} C_VEL
LIN {X 0,Y 594.37,Z 369.071,A -85,B 0,C 180,E1 -1126.16,E2 -1126.16} C_VEL
LIN {X 0,Y 594.383,Z 369.075,A -85,B 0,C 180,E1 -1128.536,E2 -1128.536} C_VEL
LIN {X 0,Y 594.412,Z 369.108,A -85,B 0,C 180,E1 -1131.352,E2 -1131.352} C_VEL
LIN {X 0,Y 594.427,Z 374.346,A -85,B 0,C 180,E1 -1133.761,E2 -1133.761} C_VEL
LIN {X 0,Y 594.41,Z 379.931,A -85,B 0,C 180,E1 -1136.241,E2 -1136.241} C_VEL
LIN {X 0,Y 594.397,Z 385.545,A -85,B 0,C 180,E1 -1138.651,E2 -1138.651} C_VEL
LIN {X 0,Y 594.386,Z 391.224,A -85,B 0,C 180,E1 -1141.042,E2 -1141.042} C_VEL
LIN {X 0,Y 594.348,Z 398.556,A -85,B 0,C 180,E1 -1144.054,E2 -1144.054} C_VEL
LIN {X 0,Y 594.317,Z 404.127,A -85,B 0,C 180,E1 -1146.293,E2 -1146.293} C_VEL
LIN {X 0,Y 594.346,Z 411.556,A -85,B 0,C 180,E1 -1149.222,E2 -1149.222} C_VEL
LIN {X 0,Y 594.288,Z 418.984,A -85,B 0,C 180,E1 -1152.093,E2 -1152.093} C_VEL
LIN {X 0,Y 594.258,Z 424.556,A -85,B 0,C 180,E1 -1154.216,E2 -1154.216} C_VEL
LIN {X 0,Y 594.295,Z 427.839,A -85,B 0,C 180,E1 -1155.458,E2 -1155.458} C_VEL
LIN {X 0,Y 594.872,Z 431.658,A -85,B 0,C 180,E1 -1155.533,E2 -1155.533} C_VEL
LIN {X 0,Y 594.808,Z 446.413,A -85,B 0,C 180,E1 -1155.839,E2 -1155.839} C_VEL
LIN {X 0,Y 594.735,Z 460.011,A -85,B 0,C 180,E1 -1156.264,E2 -1156.264} C_VEL
LIN {X 0,Y 594.668,Z 473.883,A -85,B 0,C 180,E1 -1156.85,E2 -1156.85} C_VEL
LIN {X 0,Y 594.597,Z 486.681,A -85,B 0,C 180,E1 -1157.543,E2 -1157.543} C_VEL
LIN {X 0,Y 594.505,Z 498.311,A -85,B 0,C 180,E1 -1158.32,E2 -1158.32} C_VEL
LIN {X 0,Y 594.475,Z 509.931,A -85,B 0,C 180,E1 -1159.269,E2 -1159.269} C_VEL
LIN {X 0,Y 594.391,Z 520.333,A -85,B 0,C 180,E1 -1160.3,E2 -1160.3} C_VEL
LIN {X 0,Y 594.355,Z 528.912,A -85,B 0,C 180,E1 -1161.329,E2 -1161.329} C_VEL
LIN {X 0,Y 594.314,Z 537.114,A -85,B 0,C 180,E1 -1162.526,E2 -1162.526} C_VEL
LIN {X 0,Y 594.271,Z 543.232,A -85,B 0,C 180,E1 -1163.619,E2 -1163.619} C_VEL
LIN {X 0,Y 594.247,Z 548.961,A -85,B 0,C 180,E1 -1164.911,E2 -1164.911} C_VEL
LIN {X 0,Y 594.259,Z 552.442,A -85,B 0,C 180,E1 -1165.931,E2 -1165.931} C_VEL
LIN {X 0,Y 594.224,Z 555.831,A -85,B 0,C 180,E1 -1167.288,E2 -1167.288} C_VEL
LIN {X 0,Y 594.242,Z 557.831,A -85,B 0,C 180,E1 -1168.645,E2 -1168.645} C_VEL
LIN {X 0,Y 594.234,Z 558.5,A -85,B 0,C 180,E1 -1170,E2 -1170} C_VEL
LIN {X 0,Y 594.242,Z 557.831,A -85,B 0,C 180,E1 -1171.355,E2 -1171.355} C_VEL
LIN {X 0,Y 594.224,Z 555.832,A -85,B 0,C 180,E1 -1172.712,E2 -1172.712} C_VEL
LIN {X 0,Y 594.259,Z 552.443,A -85,B 0,C 180,E1 -1174.069,E2 -1174.069} C_VEL
LIN {X 0,Y 594.275,Z 547.568,A -85,B 0,C 180,E1 -1175.429,E2 -1175.429} C_VEL
LIN {X 0,Y 594.3,Z 542.033,A -85,B 0,C 180,E1 -1176.607,E2 -1176.607} C_VEL
LIN {X 0,Y 594.316,Z 534.919,A -85,B 0,C 180,E1 -1177.816,E2 -1177.816} C_VEL
LIN {X 0,Y 594.369,Z 526.199,A -85,B 0,C 180,E1 -1179.014,E2 -1179.014} C_VEL
LIN {X 0,Y 594.4,Z 517.082,A -85,B 0,C 180,E1 -1180.044,E2 -1180.044} C_VEL
LIN {X 0,Y 594.479,Z 506.701,A -85,B 0,C 180,E1 -1181.018,E2 -1181.018} C_VEL
LIN {X 0,Y 594.572,Z 494.705,A -85,B 0,C 180,E1 -1181.938,E2 -1181.938} C_VEL
LIN {X 0,Y 594.61,Z 482.212,A -85,B 0,C 180,E1 -1182.717,E2 -1182.717} C_VEL
LIN {X 0,Y 594.681,Z 470.129,A -85,B 0,C 180,E1 -1183.324,E2 -1183.324} C_VEL
LIN {X 0,Y 594.778,Z 456.177,A -85,B 0,C 180,E1 -1183.866,E2 -1183.866} C_VEL
LIN {X 0,Y 594.808,Z 441.986,A -85,B 0,C 180,E1 -1184.267,E2 -1184.267} C_VEL
LIN {X 0,Y 594.704,Z 430.289,A -85,B 0,C 180,E1 -1184.491,E2 -1184.491} C_VEL
LIN {X 0,Y 594.287,Z 427.84,A -85,B 0,C 180,E1 -1184.542,E2 -1184.542} C_VEL
LIN {X 0,Y 594.297,Z 420.842,A -85,B 0,C 180,E1 -1187.196,E2 -1187.196} C_VEL
LIN {X 0,Y 594.291,Z 415.27,A -85,B 0,C 180,E1 -1189.337,E2 -1189.337} C_VEL
LIN {X 0,Y 594.308,Z 409.699,A -85,B 0,C 180,E1 -1191.506,E2 -1191.506} C_VEL
LIN {X 0,Y 594.347,Z 402.328,A -85,B 0,C 180,E1 -1194.425,E2 -1194.425} C_VEL
LIN {X 0,Y 594.362,Z 396.699,A -85,B 0,C 180,E1 -1196.701,E2 -1196.701} C_VEL
LIN {X 0,Y 594.378,Z 389.27,A -85,B 0,C 180,E1 -1199.776,E2 -1199.776} C_VEL
LIN {X 0,Y 594.393,Z 383.671,A -85,B 0,C 180,E1 -1202.146,E2 -1202.146} C_VEL
LIN {X 0,Y 594.409,Z 378.056,A -85,B 0,C 180,E1 -1204.578,E2 -1204.578} C_VEL
LIN {X 0,Y 594.441,Z 372.494,A -85,B 0,C 180,E1 -1207.083,E2 -1207.083} C_VEL
LIN {X 0,Y 594.396,Z 369.072,A -85,B 0,C 180,E1 -1208.706,E2 -1208.706} C_VEL
LIN {X 0,Y 594.383,Z 369.07,A -85,B 0,C 180,E1 -1211.848,E2 -1211.848} C_VEL
LIN {X 0,Y 594.357,Z 369.076,A -85,B 0,C 180,E1 -1214.808,E2 -1214.808} C_VEL
LIN {X 0,Y 594.368,Z 369.075,A -85,B 0,C 180,E1 -1217.625,E2 -1217.625} C_VEL
LIN {X 0,Y 594.395,Z 369.067,A -85,B 0,C 180,E1 -1220.321,E2 -1220.321} C_VEL
LIN {X 0,Y 594.387,Z 369.072,A -85,B 0,C 180,E1 -1222.913,E2 -1222.913} C_VEL
LIN {X 0,Y 594.385,Z 369.074,A -85,B 0,C 180,E1 -1225.861,E2 -1225.861} C_VEL
LIN {X 0,Y 594.372,Z 369.071,A -85,B 0,C 180,E1 -1228.65,E2 -1228.65} C_VEL
LIN {X 0,Y 594.384,Z 369.072,A -85,B 0,C 180,E1 -1231.042,E2 -1231.042} C_VEL
LIN {X 0,Y 594.386,Z 369.068,A -85,B 0,C 180,E1 -1233.301,E2 -1233.301} C_VEL
LIN {X 0,Y 594.392,Z 369.068,A -85,B 0,C 180,E1 -1236.296,E2 -1236.296} C_VEL
LIN {X 0,Y 594.401,Z 369.069,A -85,B 0,C 180,E1 -1239.224,E2 -1239.224} C_VEL
LIN {X 0,Y 594.383,Z 369.075,A -85,B 0,C 180,E1 -1242.096,E2 -1242.096} C_VEL
LIN {X 0,Y 594.368,Z 369.072,A -85,B 0,C 180,E1 -1244.219,E2 -1244.219} C_VEL
LIN {X 0,Y 594.373,Z 369.077,A -85,B 0,C 180,E1 -1247.017,E2 -1247.017} C_VEL
LIN {X 0,Y 594.396,Z 369.068,A -85,B 0,C 180,E1 -1249.784,E2 -1249.784} C_VEL
LIN {X 0,Y 594.395,Z 369.067,A -85,B 0,C 180,E1 -1252.527,E2 -1252.527} C_VEL
LIN {X 0,Y 594.399,Z 369.072,A -85,B 0,C 180,E1 -1255.252,E2 -1255.252} C_VEL
LIN {X 0,Y 594.395,Z 369.069,A -85,B 0,C 180,E1 -1257.967,E2 -1257.967} C_VEL
LIN {X 0,Y 594.42,Z 369.064,A -85,B 0,C 180,E1 -1260.677,E2 -1260.677} C_VEL
LIN {X 0,Y 594.383,Z 369.074,A -85,B 0,C 180,E1 -1263.389,E2 -1263.389} C_VEL
LIN {X 0,Y 594.365,Z 369.073,A -85,B 0,C 180,E1 -1266.109,E2 -1266.109} C_VEL
LIN {X 0,Y 594.383,Z 369.069,A -85,B 0,C 180,E1 -1268.842,E2 -1268.842} C_VEL
LIN {X 0,Y 594.394,Z 369.071,A -85,B 0,C 180,E1 -1271.596,E2 -1271.596} C_VEL
LIN {X 0,Y 594.392,Z 369.071,A -85,B 0,C 180,E1 -1274.377,E2 -1274.377} C_VEL
LIN {X 0,Y 594.361,Z 369.071,A -85,B 0,C 180,E1 -1275.329,E2 -1275.329} C_VEL
LIN {X 0,Y 593.69,Z 369.159,A -85,B 0,C 180,E1 -1275.895,E2 -1275.895} C_VEL
LIN {X 0,Y 590.838,Z 369.514,A -85,B 0,C 180,E1 -1276.813,E2 -1276.813} C_VEL
LIN {X 0,Y 588.434,Z 369.814,A -85,B 0,C 180,E1 -1277.552,E2 -1277.552} C_VEL
LIN {X 0,Y 587.406,Z 369.942,A -85,B 0,C 180,E1 -1278.122,E2 -1278.122} C_VEL
LIN {X 0,Y 587.325,Z 369.949,A -85,B 0,C 180,E1 -1278.315,E2 -1278.315} C_VEL
LIN {X 0,Y 587.333,Z 369.953,A -85,B 0,C 180,E1 -1281.038,E2 -1281.038} C_VEL
LIN {X 0,Y 587.326,Z 369.949,A -85,B 0,C 180,E1 -1283.259,E2 -1283.259} C_VEL
LIN {X 0,Y 587.334,Z 369.948,A -85,B 0,C 180,E1 -1285.517,E2 -1285.517} C_VEL
LIN {X 0,Y 587.351,Z 369.948,A -85,B 0,C 180,E1 -1287.818,E2 -1287.818} C_VEL
LIN {X 0,Y 587.339,Z 369.949,A -85,B 0,C 180,E1 -1290.51,E2 -1290.51} C_VEL
LIN {X 0,Y 587.336,Z 369.947,A -85,B 0,C 180,E1 -1293.397,E2 -1293.397} C_VEL
LIN {X 0,Y 587.359,Z 369.948,A -85,B 0,C 180,E1 -1295.895,E2 -1295.895} C_VEL
LIN {X 0,Y 587.335,Z 369.948,A -85,B 0,C 180,E1 -1298.479,E2 -1298.479} C_VEL
LIN {X 0,Y 587.337,Z 369.947,A -85,B 0,C 180,E1 -1301.157,E2 -1301.157} C_VEL
LIN {X 0,Y 587.329,Z 369.95,A -85,B 0,C 180,E1 -1304.113,E2 -1304.113} C_VEL
LIN {X 0,Y 587.327,Z 369.954,A -85,B 0,C 180,E1 -1306.995,E2 -1306.995} C_VEL
LIN {X 0,Y 587.319,Z 369.95,A -85,B 0,C 180,E1 -1309.746,E2 -1309.746} C_VEL
LIN {X 0,Y 587.316,Z 370.041,A -85,B 0,C 180,E1 -1311.52,E2 -1311.52} C_VEL
LIN {X 0,Y 587.362,Z 374.756,A -85,B 0,C 180,E1 -1314.105,E2 -1314.105} C_VEL
LIN {X 0,Y 587.344,Z 380.014,A -85,B 0,C 180,E1 -1316.888,E2 -1316.888} C_VEL
LIN {X 0,Y 587.287,Z 385.06,A -85,B 0,C 180,E1 -1319.499,E2 -1319.499} C_VEL
LIN {X 0,Y 587.275,Z 390.71,A -85,B 0,C 180,E1 -1322.322,E2 -1322.322} C_VEL
LIN {X 0,Y 587.25,Z 396.721,A -85,B 0,C 180,E1 -1325.237,E2 -1325.237} C_VEL
LIN {X 0,Y 587.248,Z 401.447,A -85,B 0,C 180,E1 -1327.482,E2 -1327.482} C_VEL
LIN {X 0,Y 587.2,Z 406.174,A -85,B 0,C 180,E1 -1329.691,E2 -1329.691} C_VEL
LIN {X 0,Y 587.177,Z 410.901,A -85,B 0,C 180,E1 -1331.869,E2 -1331.869} C_VEL
LIN {X 0,Y 587.171,Z 415.628,A -85,B 0,C 180,E1 -1334.021,E2 -1334.021} C_VEL
LIN {X 0,Y 587.216,Z 418.533,A -85,B 0,C 180,E1 -1335.333,E2 -1335.333} C_VEL
LIN {X 0,Y 587.968,Z 423.846,A -85,B 0,C 180,E1 -1335.44,E2 -1335.44} C_VEL
LIN {X 0,Y 587.903,Z 438.605,A -85,B 0,C 180,E1 -1335.778,E2 -1335.778} C_VEL
LIN {X 0,Y 587.819,Z 452.81,A -85,B 0,C 180,E1 -1336.254,E2 -1336.254} C_VEL
LIN {X 0,Y 587.693,Z 466.493,A -85,B 0,C 180,E1 -1336.867,E2 -1336.867} C_VEL
LIN {X 0,Y 587.611,Z 478.785,A -85,B 0,C 180,E1 -1337.568,E2 -1337.568} C_VEL
LIN {X 0,Y 587.534,Z 491.197,A -85,B 0,C 180,E1 -1338.442,E2 -1338.442} C_VEL
LIN {X 0,Y 587.444,Z 501.366,A -85,B 0,C 180,E1 -1339.313,E2 -1339.313} C_VEL
LIN {X 0,Y 587.323,Z 511.465,A -85,B 0,C 180,E1 -1340.356,E2 -1340.356} C_VEL
LIN {X 0,Y 587.277,Z 519.85,A -85,B 0,C 180,E1 -1341.397,E2 -1341.397} C_VEL
LIN {X 0,Y 587.245,Z 527.863,A -85,B 0,C 180,E1 -1342.608,E2 -1342.608} C_VEL
LIN {X 0,Y 587.204,Z 534.316,A -85,B 0,C 180,E1 -1343.816,E2 -1343.816} C_VEL
LIN {X 0,Y 587.158,Z 538.794,A -85,B 0,C 180,E1 -1344.85,E2 -1344.85} C_VEL
LIN {X 0,Y 587.181,Z 542.305,A -85,B 0,C 180,E1 -1345.882,E2 -1345.882} C_VEL
LIN {X 0,Y 587.13,Z 545.739,A -85,B 0,C 180,E1 -1347.256,E2 -1347.256} C_VEL
LIN {X 0,Y 587.145,Z 547.781,A -85,B 0,C 180,E1 -1348.628,E2 -1348.628} C_VEL
LIN {X 0,Y 587.136,Z 548.496,A -85,B 0,C 180,E1 -1350,E2 -1350} C_VEL
LIN {X 0,Y 587.142,Z 547.881,A -85,B 0,C 180,E1 -1351.372,E2 -1351.372} C_VEL
LIN {X 0,Y 587.128,Z 545.925,A -85,B 0,C 180,E1 -1352.744,E2 -1352.744} C_VEL
LIN {X 0,Y 587.182,Z 542.58,A -85,B 0,C 180,E1 -1354.118,E2 -1354.118} C_VEL
LIN {X 0,Y 587.2,Z 537.753,A -85,B 0,C 180,E1 -1355.495,E2 -1355.495} C_VEL
LIN {X 0,Y 587.21,Z 531.288,A -85,B 0,C 180,E1 -1356.874,E2 -1356.874} C_VEL
LIN {X 0,Y 587.269,Z 524.089,A -85,B 0,C 180,E1 -1358.084,E2 -1358.084} C_VEL
LIN {X 0,Y 587.332,Z 516.551,A -85,B 0,C 180,E1 -1359.123,E2 -1359.123} C_VEL
LIN {X 0,Y 587.376,Z 507.5,A -85,B 0,C 180,E1 -1360.165,E2 -1360.165} C_VEL
LIN {X 0,Y 587.504,Z 496.543,A -85,B 0,C 180,E1 -1361.209,E2 -1361.209} C_VEL
LIN {X 0,Y 587.577,Z 485.361,A -85,B 0,C 180,E1 -1362.082,E2 -1362.082} C_VEL
LIN {X 0,Y 587.635,Z 473.013,A -85,B 0,C 180,E1 -1362.871,E2 -1362.871} C_VEL
LIN {X 0,Y 587.769,Z 461.135,A -85,B 0,C 180,E1 -1363.483,E2 -1363.483} C_VEL
LIN {X 0,Y 587.871,Z 447.893,A -85,B 0,C 180,E1 -1364.019,E2 -1364.019} C_VEL
LIN {X 0,Y 587.924,Z 434.196,A -85,B 0,C 180,E1 -1364.429,E2 -1364.429} C_VEL
LIN {X 0,Y 587.846,Z 422.002,A -85,B 0,C 180,E1 -1364.683,E2 -1364.683} C_VEL
LIN {X 0,Y 587.213,Z 418.508,A -85,B 0,C 180,E1 -1364.769,E2 -1364.769} C_VEL
LIN {X 0,Y 587.21,Z 412.673,A -85,B 0,C 180,E1 -1367.41,E2 -1367.41} C_VEL
LIN {X 0,Y 587.204,Z 407.944,A -85,B 0,C 180,E1 -1369.58,E2 -1369.58} C_VEL
LIN {X 0,Y 587.217,Z 403.215,A -85,B 0,C 180,E1 -1371.779,E2 -1371.779} C_VEL
LIN {X 0,Y 587.245,Z 397.34,A -85,B 0,C 180,E1 -1374.557,E2 -1374.557} C_VEL
LIN {X 0,Y 587.239,Z 392.178,A -85,B 0,C 180,E1 -1377.051,E2 -1377.051} C_VEL
LIN {X 0,Y 587.269,Z 387.461,A -85,B 0,C 180,E1 -1379.384,E2 -1379.384} C_VEL
LIN {X 0,Y 587.343,Z 382.643,A -85,B 0,C 180,E1 -1381.835,E2 -1381.835} C_VEL
LIN {X 0,Y 587.359,Z 377.821,A -85,B 0,C 180,E1 -1384.349,E2 -1384.349} C_VEL
LIN {X 0,Y 587.357,Z 373.346,A -85,B 0,C 180,E1 -1386.747,E2 -1386.747} C_VEL
LIN {X 0,Y 587.311,Z 370.203,A -85,B 0,C 180,E1 -1388.481,E2 -1388.481} C_VEL
LIN {X 0,Y 587.319,Z 369.951,A -85,B 0,C 180,E1 -1390.254,E2 -1390.254} C_VEL
LIN {X 0,Y 587.329,Z 369.954,A -85,B 0,C 180,E1 -1393.119,E2 -1393.119} C_VEL
LIN {X 0,Y 587.315,Z 369.953,A -85,B 0,C 180,E1 -1396.049,E2 -1396.049} C_VEL
LIN {X 0,Y 587.338,Z 369.947,A -85,B 0,C 180,E1 -1398.925,E2 -1398.925} C_VEL
LIN {X 0,Y 587.332,Z 369.949,A -85,B 0,C 180,E1 -1401.521,E2 -1401.521} C_VEL
LIN {X 0,Y 587.356,Z 369.95,A -85,B 0,C 180,E1 -1404.455,E2 -1404.455} C_VEL
LIN {X 0,Y 587.342,Z 369.946,A -85,B 0,C 180,E1 -1406.888,E2 -1406.888} C_VEL
LIN {X 0,Y 587.336,Z 369.947,A -85,B 0,C 180,E1 -1409.83,E2 -1409.83} C_VEL
LIN {X 0,Y 587.355,Z 369.949,A -85,B 0,C 180,E1 -1412.307,E2 -1412.307} C_VEL
LIN {X 0,Y 587.355,Z 369.945,A -85,B 0,C 180,E1 -1415.242,E2 -1415.242} C_VEL
LIN {X 0,Y 587.324,Z 369.948,A -85,B 0,C 180,E1 -1418.226,E2 -1418.226} C_VEL
LIN {X 0,Y 587.349,Z 369.945,A -85,B 0,C 180,E1 -1421.151,E2 -1421.151} C_VEL
LIN {X 0,Y 587.327,Z 369.952,A -85,B 0,C 180,E1 -1424.025,E2 -1424.025} C_VEL
LIN {X 0,Y 587.362,Z 369.943,A -85,B 0,C 180,E1 -1426.154,E2 -1426.154} C_VEL
LIN {X 0,Y 587.342,Z 369.949,A -85,B 0,C 180,E1 -1428.962,E2 -1428.962} C_VEL
LIN {X 0,Y 587.369,Z 369.947,A -85,B 0,C 180,E1 -1431.745,E2 -1431.745} C_VEL
LIN {X 0,Y 587.361,Z 369.944,A -85,B 0,C 180,E1 -1434.507,E2 -1434.507} C_VEL
LIN {X 0,Y 587.378,Z 369.943,A -85,B 0,C 180,E1 -1437.257,E2 -1437.257} C_VEL
LIN {X 0,Y 587.384,Z 369.947,A -85,B 0,C 180,E1 -1440,E2 -1440} C_VEL
LIN {X 0,Y 587.379,Z 369.942,A -85,B 0,C 180,E1 -1442.743,E2 -1442.743} C_VEL
LIN {X 0,Y 587.358,Z 369.944,A -85,B 0,C 180,E1 -1445.493,E2 -1445.493} C_VEL
LIN {X 0,Y 587.345,Z 369.951,A -85,B 0,C 180,E1 -1448.256,E2 -1448.256} C_VEL
LIN {X 0,Y 587.352,Z 369.948,A -85,B 0,C 180,E1 -1451.134,E2 -1451.134} C_VEL
LIN {X 0,Y 587.369,Z 369.945,A -85,B 0,C 180,E1 -1454.26,E2 -1454.26} C_VEL
LIN {X 0,Y 587.359,Z 369.945,A -85,B 0,C 180,E1 -1457.406,E2 -1457.406} C_VEL
LIN {X 0,Y 587.331,Z 369.947,A -85,B 0,C 180,E1 -1460.305,E2 -1460.305} C_VEL
LIN {X 0,Y 587.326,Z 369.948,A -85,B 0,C 180,E1 -1463.259,E2 -1463.259} C_VEL
LIN {X 0,Y 587.332,Z 369.948,A -85,B 0,C 180,E1 -1465.517,E2 -1465.517} C_VEL
LIN {X 0,Y 587.351,Z 369.948,A -85,B 0,C 180,E1 -1467.818,E2 -1467.818} C_VEL
LIN {X 0,Y 587.34,Z 369.948,A -85,B 0,C 180,E1 -1470.51,E2 -1470.51} C_VEL
LIN {X 0,Y 587.336,Z 369.947,A -85,B 0,C 180,E1 -1473.397,E2 -1473.397} C_VEL
LIN {X 0,Y 587.359,Z 369.948,A -85,B 0,C 180,E1 -1475.895,E2 -1475.895} C_VEL
LIN {X 0,Y 587.335,Z 369.948,A -85,B 0,C 180,E1 -1478.479,E2 -1478.479} C_VEL
LIN {X 0,Y 587.338,Z 369.947,A -85,B 0,C 180,E1 -1481.157,E2 -1481.157} C_VEL
LIN {X 0,Y 587.314,Z 369.952,A -85,B 0,C 180,E1 -1484.112,E2 -1484.112} C_VEL
LIN {X 0,Y 587.32,Z 369.955,A -85,B 0,C 180,E1 -1486.994,E2 -1486.994} C_VEL
LIN {X 0,Y 587.321,Z 369.95,A -85,B 0,C 180,E1 -1489.746,E2 -1489.746} C_VEL
LIN {X 0,Y 587.383,Z 370.126,A -85,B 0,C 180,E1 -1491.294,E2 -1491.294} C_VEL
LIN {X 0,Y 587.434,Z 374.382,A -85,B 0,C 180,E1 -1493.281,E2 -1493.281} C_VEL
LIN {X 0,Y 587.394,Z 379.896,A -85,B 0,C 180,E1 -1495.782,E2 -1495.782} C_VEL
LIN {X 0,Y 587.364,Z 385.517,A -85,B 0,C 180,E1 -1498.232,E2 -1498.232} C_VEL
LIN {X 0,Y 587.352,Z 391.705,A -85,B 0,C 180,E1 -1500.866,E2 -1500.866} C_VEL
LIN {X 0,Y 587.31,Z 398.821,A -85,B 0,C 180,E1 -1503.829,E2 -1503.829} C_VEL
LIN {X 0,Y 587.253,Z 404.127,A -85,B 0,C 180,E1 -1505.99,E2 -1505.99} C_VEL
LIN {X 0,Y 587.258,Z 409.699,A -85,B 0,C 180,E1 -1508.223,E2 -1508.223} C_VEL
LIN {X 0,Y 587.256,Z 417.127,A -85,B 0,C 180,E1 -1511.148,E2 -1511.148} C_VEL
LIN {X 0,Y 587.191,Z 424.556,A -85,B 0,C 180,E1 -1514.021,E2 -1514.021} C_VEL
LIN {X 0,Y 587.206,Z 427.834,A -85,B 0,C 180,E1 -1515.277,E2 -1515.277} C_VEL
LIN {X 0,Y 588.002,Z 432.966,A -85,B 0,C 180,E1 -1515.38,E2 -1515.38} C_VEL
LIN {X 0,Y 587.907,Z 447.689,A -85,B 0,C 180,E1 -1515.706,E2 -1515.706} C_VEL
LIN {X 0,Y 587.799,Z 461.711,A -85,B 0,C 180,E1 -1516.165,E2 -1516.165} C_VEL
LIN {X 0,Y 587.718,Z 475.635,A -85,B 0,C 180,E1 -1516.779,E2 -1516.779} C_VEL
LIN {X 0,Y 587.623,Z 488.094,A -85,B 0,C 180,E1 -1517.48,E2 -1517.48} C_VEL
LIN {X 0,Y 587.513,Z 499.474,A -85,B 0,C 180,E1 -1518.266,E2 -1518.266} C_VEL
LIN {X 0,Y 587.467,Z 509.932,A -85,B 0,C 180,E1 -1519.139,E2 -1519.139} C_VEL
LIN {X 0,Y 587.353,Z 520.333,A -85,B 0,C 180,E1 -1520.182,E2 -1520.182} C_VEL
LIN {X 0,Y 587.311,Z 528.912,A -85,B 0,C 180,E1 -1521.224,E2 -1521.224} C_VEL
LIN {X 0,Y 587.249,Z 537.114,A -85,B 0,C 180,E1 -1522.435,E2 -1522.435} C_VEL
LIN {X 0,Y 587.18,Z 543.679,A -85,B 0,C 180,E1 -1523.635,E2 -1523.635} C_VEL
LIN {X 0,Y 587.16,Z 548.961,A -85,B 0,C 180,E1 -1524.849,E2 -1524.849} C_VEL
LIN {X 0,Y 587.179,Z 552.442,A -85,B 0,C 180,E1 -1525.882,E2 -1525.882} C_VEL
LIN {X 0,Y 587.13,Z 555.831,A -85,B 0,C 180,E1 -1527.256,E2 -1527.256} C_VEL
LIN {X 0,Y 587.142,Z 557.831,A -85,B 0,C 180,E1 -1528.628,E2 -1528.628} C_VEL
LIN {X 0,Y 587.135,Z 558.5,A -85,B 0,C 180,E1 -1530,E2 -1530} C_VEL
LIN {X 0,Y 587.142,Z 557.832,A -85,B 0,C 180,E1 -1531.372,E2 -1531.372} C_VEL
LIN {X 0,Y 587.13,Z 555.832,A -85,B 0,C 180,E1 -1532.744,E2 -1532.744} C_VEL
LIN {X 0,Y 587.179,Z 552.443,A -85,B 0,C 180,E1 -1534.118,E2 -1534.118} C_VEL
LIN {X 0,Y 587.2,Z 547.568,A -85,B 0,C 180,E1 -1535.494,E2 -1535.494} C_VEL
LIN {X 0,Y 587.209,Z 541.052,A -85,B 0,C 180,E1 -1536.874,E2 -1536.874} C_VEL
LIN {X 0,Y 587.268,Z 533.799,A -85,B 0,C 180,E1 -1538.083,E2 -1538.083} C_VEL
LIN {X 0,Y 587.321,Z 524.823,A -85,B 0,C 180,E1 -1539.296,E2 -1539.296} C_VEL
LIN {X 0,Y 587.372,Z 515.391,A -85,B 0,C 180,E1 -1540.339,E2 -1540.339} C_VEL
LIN {X 0,Y 587.475,Z 505.025,A -85,B 0,C 180,E1 -1541.29,E2 -1541.29} C_VEL
LIN {X 0,Y 587.574,Z 493.43,A -85,B 0,C 180,E1 -1542.17,E2 -1542.17} C_VEL
LIN {X 0,Y 587.665,Z 480.648,A -85,B 0,C 180,E1 -1542.958,E2 -1542.958} C_VEL
LIN {X 0,Y 587.77,Z 468.161,A -85,B 0,C 180,E1 -1543.571,E2 -1543.571} C_VEL
LIN {X 0,Y 587.892,Z 454.961,A -85,B 0,C 180,E1 -1544.074,E2 -1544.074} C_VEL
LIN {X 0,Y 587.958,Z 441.203,A -85,B 0,C 180,E1 -1544.455,E2 -1544.455} C_VEL
LIN {X 0,Y 587.822,Z 431.138,A -85,B 0,C 180,E1 -1544.652,E2 -1544.652} C_VEL
LIN {X 0,Y 587.201,Z 427.806,A -85,B 0,C 180,E1 -1544.734,E2 -1544.734} C_VEL
LIN {X 0,Y 587.22,Z 420.842,A -85,B 0,C 180,E1 -1547.41,E2 -1547.41} C_VEL
LIN {X 0,Y 587.218,Z 415.27,A -85,B 0,C 180,E1 -1549.579,E2 -1549.579} C_VEL
LIN {X 0,Y 587.257,Z 409.699,A -85,B 0,C 180,E1 -1551.777,E2 -1551.777} C_VEL
LIN {X 0,Y 587.282,Z 402.755,A -85,B 0,C 180,E1 -1554.565,E2 -1554.565} C_VEL
LIN {X 0,Y 587.312,Z 396.699,A -85,B 0,C 180,E1 -1557.047,E2 -1557.047} C_VEL
LIN {X 0,Y 587.348,Z 391.117,A -85,B 0,C 180,E1 -1559.379,E2 -1559.379} C_VEL
LIN {X 0,Y 587.365,Z 385.342,A -85,B 0,C 180,E1 -1561.839,E2 -1561.839} C_VEL
LIN {X 0,Y 587.382,Z 379.597,A -85,B 0,C 180,E1 -1564.352,E2 -1564.352} C_VEL
LIN {X 0,Y 587.433,Z 374.335,A -85,B 0,C 180,E1 -1566.741,E2 -1566.741} C_VEL
LIN {X 0,Y 587.344,Z 369.951,A -85,B 0,C 180,E1 -1568.839,E2 -1568.839} C_VEL
LIN {X 0,Y 587.338,Z 369.953,A -85,B 0,C 180,E1 -1571.157,E2 -1571.157} C_VEL
LIN {X 0,Y 587.328,Z 369.949,A -85,B 0,C 180,E1 -1574.113,E2 -1574.113} C_VEL
LIN {X 0,Y 587.314,Z 369.95,A -85,B 0,C 180,E1 -1576.993,E2 -1576.993} C_VEL
LIN {X 0,Y 587.322,Z 369.951,A -85,B 0,C 180,E1 -1579.746,E2 -1579.746} C_VEL
LIN {X 0,Y 587.347,Z 369.948,A -85,B 0,C 180,E1 -1582.392,E2 -1582.392} C_VEL
LIN {X 0,Y 587.351,Z 369.945,A -85,B 0,C 180,E1 -1584.946,E2 -1584.946} C_VEL
LIN {X 0,Y 587.341,Z 369.951,A -85,B 0,C 180,E1 -1587.421,E2 -1587.421} C_VEL
LIN {X 0,Y 587.336,Z 369.947,A -85,B 0,C 180,E1 -1589.83,E2 -1589.83} C_VEL
LIN {X 0,Y 587.354,Z 369.949,A -85,B 0,C 180,E1 -1592.307,E2 -1592.307} C_VEL
LIN {X 0,Y 587.353,Z 369.946,A -85,B 0,C 180,E1 -1595.242,E2 -1595.242} C_VEL
LIN {X 0,Y 587.323,Z 369.948,A -85,B 0,C 180,E1 -1598.226,E2 -1598.226} C_VEL
LIN {X 0,Y 587.349,Z 369.945,A -85,B 0,C 180,E1 -1601.151,E2 -1601.151} C_VEL
LIN {X 0,Y 587.349,Z 369.946,A -85,B 0,C 180,E1 -1603.311,E2 -1603.311} C_VEL
LIN {X 0,Y 587.363,Z 369.943,A -85,B 0,C 180,E1 -1606.154,E2 -1606.154} C_VEL
LIN {X 0,Y 587.341,Z 369.948,A -85,B 0,C 180,E1 -1608.962,E2 -1608.962} C_VEL
LIN {X 0,Y 587.366,Z 369.947,A -85,B 0,C 180,E1 -1611.745,E2 -1611.745} C_VEL
LIN {X 0,Y 587.358,Z 369.944,A -85,B 0,C 180,E1 -1614.507,E2 -1614.507} C_VEL
LIN {X 0,Y 587.379,Z 369.942,A -85,B 0,C 180,E1 -1617.257,E2 -1617.257} C_VEL
LIN {X 0,Y 587.386,Z 369.947,A -85,B 0,C 180,E1 -1620,E2 -1620} C_VEL
LIN {X 0,Y 587.377,Z 369.942,A -85,B 0,C 180,E1 -1622.743,E2 -1622.743} C_VEL
LIN {X 0,Y 587.361,Z 369.944,A -85,B 0,C 180,E1 -1625.493,E2 -1625.493} C_VEL
LIN {X 0,Y 587.368,Z 369.948,A -85,B 0,C 180,E1 -1628.255,E2 -1628.255} C_VEL
LIN {X 0,Y 587.351,Z 369.948,A -85,B 0,C 180,E1 -1631.134,E2 -1631.134} C_VEL
LIN {X 0,Y 587.367,Z 369.944,A -85,B 0,C 180,E1 -1634.26,E2 -1634.26} C_VEL
LIN {X 0,Y 587.358,Z 369.945,A -85,B 0,C 180,E1 -1637.406,E2 -1637.406} C_VEL
LIN {X 0,Y 587.325,Z 369.949,A -85,B 0,C 180,E1 -1638.315,E2 -1638.315} C_VEL
LIN {X 0,Y 586.671,Z 370.03,A -85,B 0,C 180,E1 -1638.887,E2 -1638.887} C_VEL
LIN {X 0,Y 583.84,Z 370.387,A -85,B 0,C 180,E1 -1639.816,E2 -1639.816} C_VEL
LIN {X 0,Y 581.431,Z 370.69,A -85,B 0,C 180,E1 -1640.562,E2 -1640.562} C_VEL
LIN {X 0,Y 580.38,Z 370.82,A -85,B 0,C 180,E1 -1641.139,E2 -1641.139} C_VEL
LIN {X 0,Y 580.285,Z 370.828,A -85,B 0,C 180,E1 -1641.334,E2 -1641.334} C_VEL
LIN {X 0,Y 580.304,Z 370.829,A -85,B 0,C 180,E1 -1644.316,E2 -1644.316} C_VEL
LIN {X 0,Y 580.279,Z 370.826,A -85,B 0,C 180,E1 -1646.623,E2 -1646.623} C_VEL
LIN {X 0,Y 580.303,Z 370.828,A -85,B 0,C 180,E1 -1649.31,E2 -1649.31} C_VEL
LIN {X 0,Y 580.301,Z 370.826,A -85,B 0,C 180,E1 -1652.201,E2 -1652.201} C_VEL
LIN {X 0,Y 580.303,Z 370.823,A -85,B 0,C 180,E1 -1654.695,E2 -1654.695} C_VEL
LIN {X 0,Y 580.303,Z 370.829,A -85,B 0,C 180,E1 -1657.268,E2 -1657.268} C_VEL
LIN {X 0,Y 580.299,Z 370.826,A -85,B 0,C 180,E1 -1660.271,E2 -1660.271} C_VEL
LIN {X 0,Y 580.28,Z 370.827,A -85,B 0,C 180,E1 -1662.706,E2 -1662.706} C_VEL
LIN {X 0,Y 580.277,Z 370.831,A -85,B 0,C 180,E1 -1665.609,E2 -1665.609} C_VEL
LIN {X 0,Y 580.316,Z 370.823,A -85,B 0,C 180,E1 -1668.234,E2 -1668.234} C_VEL
LIN {X 0,Y 580.28,Z 370.829,A -85,B 0,C 180,E1 -1670.965,E2 -1670.965} C_VEL
LIN {X 0,Y 580.333,Z 371.753,A -85,B 0,C 180,E1 -1671.922,E2 -1671.922} C_VEL
LIN {X 0,Y 580.316,Z 376.352,A -85,B 0,C 180,E1 -1674.457,E2 -1674.457} C_VEL
LIN {X 0,Y 580.293,Z 381.06,A -85,B 0,C 180,E1 -1676.975,E2 -1676.975} C_VEL
LIN {X 0,Y 580.253,Z 385.747,A -85,B 0,C 180,E1 -1679.423,E2 -1679.423} C_VEL
LIN {X 0,Y 580.223,Z 391.118,A -85,B 0,C 180,E1 -1682.156,E2 -1682.156} C_VEL
LIN {X 0,Y 580.181,Z 396.722,A -85,B 0,C 180,E1 -1684.914,E2 -1684.914} C_VEL
LIN {X 0,Y 580.152,Z 403.024,A -85,B 0,C 180,E1 -1687.943,E2 -1687.943} C_VEL
LIN {X 0,Y 580.164,Z 409.326,A -85,B 0,C 180,E1 -1690.909,E2 -1690.909} C_VEL
LIN {X 0,Y 580.103,Z 415.629,A -85,B 0,C 180,E1 -1693.821,E2 -1693.821} C_VEL
LIN {X 0,Y 580.13,Z 418.534,A -85,B 0,C 180,E1 -1695.15,E2 -1695.15} C_VEL
LIN {X 0,Y 581.13,Z 425.015,A -85,B 0,C 180,E1 -1695.288,E2 -1695.288} C_VEL
LIN {X 0,Y 581.001,Z 439.511,A -85,B 0,C 180,E1 -1695.631,E2 -1695.631} C_VEL
LIN {X 0,Y 580.902,Z 453.947,A -85,B 0,C 180,E1 -1696.131,E2 -1696.131} C_VEL
LIN {X 0,Y 580.772,Z 466.506,A -85,B 0,C 180,E1 -1696.708,E2 -1696.708} C_VEL
LIN {X 0,Y 580.658,Z 478.796,A -85,B 0,C 180,E1 -1697.416,E2 -1697.416} C_VEL
LIN {X 0,Y 580.54,Z 491.204,A -85,B 0,C 180,E1 -1698.301,E2 -1698.301} C_VEL
LIN {X 0,Y 580.442,Z 501.394,A -85,B 0,C 180,E1 -1699.185,E2 -1699.185} C_VEL
LIN {X 0,Y 580.28,Z 511.47,A -85,B 0,C 180,E1 -1700.238,E2 -1700.238} C_VEL
LIN {X 0,Y 580.241,Z 519.854,A -85,B 0,C 180,E1 -1701.292,E2 -1701.292} C_VEL
LIN {X 0,Y 580.166,Z 527.867,A -85,B 0,C 180,E1 -1702.518,E2 -1702.518} C_VEL
LIN {X 0,Y 580.104,Z 534.319,A -85,B 0,C 180,E1 -1703.74,E2 -1703.74} C_VEL
LIN {X 0,Y 580.077,Z 538.796,A -85,B 0,C 180,E1 -1704.787,E2 -1704.787} C_VEL
LIN {X 0,Y 580.103,Z 542.307,A -85,B 0,C 180,E1 -1705.832,E2 -1705.832} C_VEL
LIN {X 0,Y 580.041,Z 545.74,A -85,B 0,C 180,E1 -1707.222,E2 -1707.222} C_VEL
LIN {X 0,Y 580.045,Z 547.782,A -85,B 0,C 180,E1 -1708.612,E2 -1708.612} C_VEL
LIN {X 0,Y 580.037,Z 548.496,A -85,B 0,C 180,E1 -1710,E2 -1710} C_VEL
LIN {X 0,Y 580.042,Z 547.88,A -85,B 0,C 180,E1 -1711.389,E2 -1711.389} C_VEL
LIN {X 0,Y 580.039,Z 545.924,A -85,B 0,C 180,E1 -1712.778,E2 -1712.778} C_VEL
LIN {X 0,Y 580.104,Z 542.579,A -85,B 0,C 180,E1 -1714.169,E2 -1714.169} C_VEL
LIN {X 0,Y 580.129,Z 537.751,A -85,B 0,C 180,E1 -1715.562,E2 -1715.562} C_VEL
LIN {X 0,Y 580.142,Z 531.285,A -85,B 0,C 180,E1 -1716.958,E2 -1716.958} C_VEL
LIN {X 0,Y 580.193,Z 524.086,A -85,B 0,C 180,E1 -1718.183,E2 -1718.183} C_VEL
LIN {X 0,Y 580.284,Z 516.547,A -85,B 0,C 180,E1 -1719.235,E2 -1719.235} C_VEL
LIN {X 0,Y 580.347,Z 507.495,A -85,B 0,C 180,E1 -1720.29,E2 -1720.29} C_VEL
LIN {X 0,Y 580.494,Z 496.537,A -85,B 0,C 180,E1 -1721.346,E2 -1721.346} C_VEL
LIN {X 0,Y 580.585,Z 485.354,A -85,B 0,C 180,E1 -1722.23,E2 -1722.23} C_VEL
LIN {X 0,Y 580.695,Z 473.005,A -85,B 0,C 180,E1 -1723.027,E2 -1723.027} C_VEL
LIN {X 0,Y 580.854,Z 461.125,A -85,B 0,C 180,E1 -1723.647,E2 -1723.647} C_VEL
LIN {X 0,Y 580.976,Z 448.241,A -85,B 0,C 180,E1 -1724.177,E2 -1724.177} C_VEL
LIN {X 0,Y 581.06,Z 434.124,A -85,B 0,C 180,E1 -1724.604,E2 -1724.604} C_VEL
LIN {X 0,Y 580.928,Z 422.701,A -85,B 0,C 180,E1 -1724.851,E2 -1724.851} C_VEL
LIN {X 0,Y 580.122,Z 418.534,A -85,B 0,C 180,E1 -1724.941,E2 -1724.941} C_VEL
LIN {X 0,Y 580.12,Z 412.672,A -85,B 0,C 180,E1 -1727.63,E2 -1727.63} C_VEL
LIN {X 0,Y 580.113,Z 407.943,A -85,B 0,C 180,E1 -1729.829,E2 -1729.829} C_VEL
LIN {X 0,Y 580.153,Z 403.213,A -85,B 0,C 180,E1 -1732.058,E2 -1732.058} C_VEL
LIN {X 0,Y 580.182,Z 396.907,A -85,B 0,C 180,E1 -1735.086,E2 -1735.086} C_VEL
LIN {X 0,Y 580.224,Z 391.304,A -85,B 0,C 180,E1 -1737.844,E2 -1737.844} C_VEL
LIN {X 0,Y 580.238,Z 385.721,A -85,B 0,C 180,E1 -1740.686,E2 -1740.686} C_VEL
LIN {X 0,Y 580.293,Z 380.681,A -85,B 0,C 180,E1 -1743.314,E2 -1743.314} C_VEL
LIN {X 0,Y 580.331,Z 376.097,A -85,B 0,C 180,E1 -1745.768,E2 -1745.768} C_VEL
LIN {X 0,Y 580.33,Z 371.798,A -85,B 0,C 180,E1 -1748.143,E2 -1748.143} C_VEL
LIN {X 0,Y 580.298,Z 370.827,A -85,B 0,C 180,E1 -1749.185,E2 -1749.185} C_VEL
LIN {X 0,Y 580.293,Z 370.827,A -85,B 0,C 180,E1 -1751.768,E2 -1751.768} C_VEL
LIN {X 0,Y 580.272,Z 370.834,A -85,B 0,C 180,E1 -1754.626,E2 -1754.626} C_VEL
LIN {X 0,Y 580.289,Z 370.828,A -85,B 0,C 180,E1 -1757.628,E2 -1757.628} C_VEL
LIN {X 0,Y 580.288,Z 370.825,A -85,B 0,C 180,E1 -1760.067,E2 -1760.067} C_VEL
LIN {X 0,Y 580.306,Z 370.825,A -85,B 0,C 180,E1 -1763.065,E2 -1763.065} C_VEL
LIN {X 0,Y 580.307,Z 370.823,A -85,B 0,C 180,E1 -1765.441,E2 -1765.441} C_VEL
LIN {X 0,Y 580.306,Z 370.824,A -85,B 0,C 180,E1 -1767.969,E2 -1767.969} C_VEL
LIN {X 0,Y 580.304,Z 370.827,A -85,B 0,C 180,E1 -1770.69,E2 -1770.69} C_VEL
LIN {X 0,Y 580.295,Z 370.825,A -85,B 0,C 180,E1 -1773.666,E2 -1773.666} C_VEL
LIN {X 0,Y 580.305,Z 370.829,A -85,B 0,C 180,E1 -1775.684,E2 -1775.684} C_VEL
LIN {X 0,Y 580.275,Z 370.826,A -85,B 0,C 180,E1 -1777.947,E2 -1777.947} C_VEL
LIN {X 0,Y 580.303,Z 370.825,A -85,B 0,C 180,E1 -1780.913,E2 -1780.913} C_VEL
LIN {X 0,Y 580.281,Z 370.832,A -85,B 0,C 180,E1 -1783.826,E2 -1783.826} C_VEL
LIN {X 0,Y 580.329,Z 370.82,A -85,B 0,C 180,E1 -1785.983,E2 -1785.983} C_VEL
LIN {X 0,Y 580.309,Z 370.827,A -85,B 0,C 180,E1 -1788.827,E2 -1788.827} C_VEL
LIN {X 0,Y 580.331,Z 370.822,A -85,B 0,C 180,E1 -1791.644,E2 -1791.644} C_VEL
LIN {X 0,Y 580.326,Z 370.82,A -85,B 0,C 180,E1 -1794.44,E2 -1794.44} C_VEL
LIN {X 0,Y 580.344,Z 370.819,A -85,B 0,C 180,E1 -1797.223,E2 -1797.223} C_VEL
LIN {X 0,Y 580.354,Z 370.823,A -85,B 0,C 180,E1 -1800,E2 -1800} C_VEL
LIN {X 0,Y 580.345,Z 370.818,A -85,B 0,C 180,E1 -1802.776,E2 -1802.776} C_VEL
LIN {X 0,Y 580.324,Z 370.82,A -85,B 0,C 180,E1 -1805.56,E2 -1805.56} C_VEL
LIN {X 0,Y 580.326,Z 370.821,A -85,B 0,C 180,E1 -1807.655,E2 -1807.655} C_VEL
LIN {X 0,Y 580.304,Z 370.822,A -85,B 0,C 180,E1 -1810.467,E2 -1810.467} C_VEL
LIN {X 0,Y 580.279,Z 370.828,A -85,B 0,C 180,E1 -1813.304,E2 -1813.304} C_VEL
LIN {X 0,Y 580.297,Z 370.823,A -85,B 0,C 180,E1 -1815.453,E2 -1815.453} C_VEL
LIN {X 0,Y 580.305,Z 370.826,A -85,B 0,C 180,E1 -1817.624,E2 -1817.624} C_VEL
LIN {X 0,Y 580.308,Z 370.824,A -85,B 0,C 180,E1 -1819.822,E2 -1819.822} C_VEL
LIN {X 0,Y 580.299,Z 370.829,A -85,B 0,C 180,E1 -1822.802,E2 -1822.802} C_VEL
LIN {X 0,Y 580.308,Z 370.822,A -85,B 0,C 180,E1 -1825.08,E2 -1825.08} C_VEL
LIN {X 0,Y 580.303,Z 370.823,A -85,B 0,C 180,E1 -1828.185,E2 -1828.185} C_VEL
LIN {X 0,Y 580.288,Z 370.829,A -85,B 0,C 180,E1 -1830.695,E2 -1830.695} C_VEL
LIN {X 0,Y 580.306,Z 370.822,A -85,B 0,C 180,E1 -1833.316,E2 -1833.316} C_VEL
LIN {X 0,Y 580.328,Z 370.826,A -85,B 0,C 180,E1 -1835.767,E2 -1835.767} C_VEL
LIN {X 0,Y 580.292,Z 370.825,A -85,B 0,C 180,E1 -1838.146,E2 -1838.146} C_VEL
LIN {X 0,Y 580.302,Z 370.826,A -85,B 0,C 180,E1 -1840.843,E2 -1840.843} C_VEL
LIN {X 0,Y 580.275,Z 370.832,A -85,B 0,C 180,E1 -1843.658,E2 -1843.658} C_VEL
LIN {X 0,Y 580.281,Z 370.828,A -85,B 0,C 180,E1 -1846.609,E2 -1846.609} C_VEL
LIN {X 0,Y 580.302,Z 370.825,A -85,B 0,C 180,E1 -1849.157,E2 -1849.157} C_VEL
LIN {X 0,Y 580.331,Z 370.943,A -85,B 0,C 180,E1 -1851.136,E2 -1851.136} C_VEL
LIN {X 0,Y 580.405,Z 374.981,A -85,B 0,C 180,E1 -1853.052,E2 -1853.052} C_VEL
LIN {X 0,Y 580.376,Z 380.146,A -85,B 0,C 180,E1 -1855.431,E2 -1855.431} C_VEL
LIN {X 0,Y 580.322,Z 385.857,A -85,B 0,C 180,E1 -1857.966,E2 -1857.966} C_VEL
LIN {X 0,Y 580.303,Z 392.185,A -85,B 0,C 180,E1 -1860.69,E2 -1860.69} C_VEL
LIN {X 0,Y 580.259,Z 399.268,A -85,B 0,C 180,E1 -1863.673,E2 -1863.673} C_VEL
LIN {X 0,Y 580.183,Z 405.984,A -85,B 0,C 180,E1 -1866.438,E2 -1866.438} C_VEL
LIN {X 0,Y 580.225,Z 411.961,A -85,B 0,C 180,E1 -1868.854,E2 -1868.854} C_VEL
LIN {X 0,Y 580.147,Z 418.984,A -85,B 0,C 180,E1 -1871.641,E2 -1871.641} C_VEL
LIN {X 0,Y 580.128,Z 424.556,A -85,B 0,C 180,E1 -1873.821,E2 -1873.821} C_VEL
LIN {X 0,Y 580.136,Z 427.849,A -85,B 0,C 180,E1 -1875.099,E2 -1875.099} C_VEL
LIN {X 0,Y 581.139,Z 433.879,A -85,B 0,C 180,E1 -1875.221,E2 -1875.221} C_VEL
LIN {X 0,Y 581.013,Z 448.122,A -85,B 0,C 180,E1 -1875.545,E2 -1875.545} C_VEL
LIN {X 0,Y 580.889,Z 461.709,A -85,B 0,C 180,E1 -1875.997,E2 -1875.997} C_VEL
LIN {X 0,Y 580.779,Z 475.637,A -85,B 0,C 180,E1 -1876.619,E2 -1876.619} C_VEL
LIN {X 0,Y 580.654,Z 488.096,A -85,B 0,C 180,E1 -1877.327,E2 -1877.327} C_VEL
LIN {X 0,Y 580.544,Z 499.475,A -85,B 0,C 180,E1 -1878.124,E2 -1878.124} C_VEL
LIN {X 0,Y 580.462,Z 509.971,A -85,B 0,C 180,E1 -1879.01,E2 -1879.01} C_VEL
LIN {X 0,Y 580.312,Z 520.333,A -85,B 0,C 180,E1 -1880.062,E2 -1880.062} C_VEL
LIN {X 0,Y 580.254,Z 528.912,A -85,B 0,C 180,E1 -1881.116,E2 -1881.116} C_VEL
LIN {X 0,Y 580.176,Z 537.115,A -85,B 0,C 180,E1 -1882.343,E2 -1882.343} C_VEL
LIN {X 0,Y 580.123,Z 542.99,A -85,B 0,C 180,E1 -1883.415,E2 -1883.415} C_VEL
LIN {X 0,Y 580.128,Z 547.568,A -85,B 0,C 180,E1 -1884.438,E2 -1884.438} C_VEL
LIN {X 0,Y 580.102,Z 552.442,A -85,B 0,C 180,E1 -1885.831,E2 -1885.831} C_VEL
LIN {X 0,Y 580.041,Z 555.831,A -85,B 0,C 180,E1 -1887.222,E2 -1887.222} C_VEL
LIN {X 0,Y 580.041,Z 557.832,A -85,B 0,C 180,E1 -1888.611,E2 -1888.611} C_VEL
LIN {X 0,Y 580.036,Z 558.5,A -85,B 0,C 180,E1 -1890,E2 -1890} C_VEL
LIN {X 0,Y 580.041,Z 557.832,A -85,B 0,C 180,E1 -1891.389,E2 -1891.389} C_VEL
LIN {X 0,Y 580.041,Z 555.833,A -85,B 0,C 180,E1 -1892.778,E2 -1892.778} C_VEL
LIN {X 0,Y 580.102,Z 552.444,A -85,B 0,C 180,E1 -1894.168,E2 -1894.168} C_VEL
LIN {X 0,Y 580.128,Z 547.568,A -85,B 0,C 180,E1 -1895.562,E2 -1895.562} C_VEL
LIN {X 0,Y 580.141,Z 541.052,A -85,B 0,C 180,E1 -1896.958,E2 -1896.958} C_VEL
LIN {X 0,Y 580.192,Z 533.8,A -85,B 0,C 180,E1 -1898.183,E2 -1898.183} C_VEL
LIN {X 0,Y 580.284,Z 524.823,A -85,B 0,C 180,E1 -1899.41,E2 -1899.41} C_VEL
LIN {X 0,Y 580.356,Z 515.392,A -85,B 0,C 180,E1 -1900.466,E2 -1900.466} C_VEL
LIN {X 0,Y 580.475,Z 505.318,A -85,B 0,C 180,E1 -1901.404,E2 -1901.404} C_VEL
LIN {X 0,Y 580.595,Z 493.431,A -85,B 0,C 180,E1 -1902.319,E2 -1902.319} C_VEL
LIN {X 0,Y 580.723,Z 480.648,A -85,B 0,C 180,E1 -1903.115,E2 -1903.115} C_VEL
LIN {X 0,Y 580.861,Z 468.159,A -85,B 0,C 180,E1 -1903.736,E2 -1903.736} C_VEL
LIN {X 0,Y 581.005,Z 455.524,A -85,B 0,C 180,E1 -1904.224,E2 -1904.224} C_VEL
LIN {X 0,Y 581.094,Z 441.707,A -85,B 0,C 180,E1 -1904.618,E2 -1904.618} C_VEL
LIN {X 0,Y 580.921,Z 432.071,A -85,B 0,C 180,E1 -1904.816,E2 -1904.816} C_VEL
LIN {X 0,Y 580.135,Z 427.806,A -85,B 0,C 180,E1 -1904.918,E2 -1904.918} C_VEL
LIN {X 0,Y 580.15,Z 420.842,A -85,B 0,C 180,E1 -1907.629,E2 -1907.629} C_VEL
LIN {X 0,Y 580.165,Z 415.27,A -85,B 0,C 180,E1 -1909.827,E2 -1909.827} C_VEL
LIN {X 0,Y 580.205,Z 409.699,A -85,B 0,C 180,E1 -1912.055,E2 -1912.055} C_VEL
LIN {X 0,Y 580.234,Z 402.27,A -85,B 0,C 180,E1 -1915.083,E2 -1915.083} C_VEL
LIN {X 0,Y 580.247,Z 395.635,A -85,B 0,C 180,E1 -1917.849,E2 -1917.849} C_VEL
LIN {X 0,Y 580.304,Z 389.213,A -85,B 0,C 180,E1 -1920.574,E2 -1920.574} C_VEL
LIN {X 0,Y 580.364,Z 382.912,A -85,B 0,C 180,E1 -1923.325,E2 -1923.325} C_VEL
LIN {X 0,Y 580.407,Z 377.504,A -85,B 0,C 180,E1 -1925.778,E2 -1925.778} C_VEL
LIN {X 0,Y 580.425,Z 371.524,A -85,B 0,C 180,E1 -1928.578,E2 -1928.578} C_VEL
LIN {X 0,Y 580.29,Z 370.83,A -85,B 0,C 180,E1 -1929.034,E2 -1929.034} C_VEL
LIN {X 0,Y 580.316,Z 370.824,A -85,B 0,C 180,E1 -1931.766,E2 -1931.766} C_VEL
LIN {X 0,Y 580.262,Z 370.835,A -85,B 0,C 180,E1 -1934.627,E2 -1934.627} C_VEL
LIN {X 0,Y 580.287,Z 370.829,A -85,B 0,C 180,E1 -1937.628,E2 -1937.628} C_VEL
LIN {X 0,Y 580.297,Z 370.824,A -85,B 0,C 180,E1 -1940.067,E2 -1940.067} C_VEL
LIN {X 0,Y 580.304,Z 370.825,A -85,B 0,C 180,E1 -1943.065,E2 -1943.065} C_VEL
LIN {X 0,Y 580.305,Z 370.824,A -85,B 0,C 180,E1 -1945.441,E2 -1945.441} C_VEL
LIN {X 0,Y 580.305,Z 370.824,A -85,B 0,C 180,E1 -1947.969,E2 -1947.969} C_VEL
LIN {X 0,Y 580.303,Z 370.828,A -85,B 0,C 180,E1 -1950.69,E2 -1950.69} C_VEL
LIN {X 0,Y 580.292,Z 370.826,A -85,B 0,C 180,E1 -1953.666,E2 -1953.666} C_VEL
LIN {X 0,Y 580.303,Z 370.83,A -85,B 0,C 180,E1 -1955.684,E2 -1955.684} C_VEL
LIN {X 0,Y 580.274,Z 370.826,A -85,B 0,C 180,E1 -1957.947,E2 -1957.947} C_VEL
LIN {X 0,Y 580.302,Z 370.825,A -85,B 0,C 180,E1 -1960.914,E2 -1960.914} C_VEL
LIN {X 0,Y 580.31,Z 370.822,A -85,B 0,C 180,E1 -1963.103,E2 -1963.103} C_VEL
LIN {X 0,Y 580.329,Z 370.82,A -85,B 0,C 180,E1 -1965.983,E2 -1965.983} C_VEL
LIN {X 0,Y 580.307,Z 370.826,A -85,B 0,C 180,E1 -1968.827,E2 -1968.827} C_VEL
LIN {X 0,Y 580.33,Z 370.823,A -85,B 0,C 180,E1 -1971.644,E2 -1971.644} C_VEL
LIN {X 0,Y 580.324,Z 370.82,A -85,B 0,C 180,E1 -1974.44,E2 -1974.44} C_VEL
LIN {X 0,Y 580.345,Z 370.819,A -85,B 0,C 180,E1 -1977.224,E2 -1977.224} C_VEL
LIN {X 0,Y 580.355,Z 370.823,A -85,B 0,C 180,E1 -1980,E2 -1980} C_VEL
LIN {X 0,Y 580.343,Z 370.819,A -85,B 0,C 180,E1 -1982.777,E2 -1982.777} C_VEL
LIN {X 0,Y 580.326,Z 370.82,A -85,B 0,C 180,E1 -1985.56,E2 -1985.56} C_VEL
LIN {X 0,Y 580.331,Z 370.823,A -85,B 0,C 180,E1 -1988.356,E2 -1988.356} C_VEL
LIN {X 0,Y 580.303,Z 370.827,A -85,B 0,C 180,E1 -1991.191,E2 -1991.191} C_VEL
LIN {X 0,Y 580.328,Z 370.819,A -85,B 0,C 180,E1 -1994.017,E2 -1994.017} C_VEL
LIN {X 0,Y 580.315,Z 370.821,A -85,B 0,C 180,E1 -1996.914,E2 -1996.914} C_VEL
LIN {X 0,Y 580.307,Z 370.824,A -85,B 0,C 180,E1 -1999.822,E2 -1999.822} C_VEL
LIN {X 0,Y 580.285,Z 370.828,A -85,B 0,C 180,E1 -2001.334,E2 -2001.334} C_VEL
LIN {X 0,Y 579.588,Z 370.913,A -85,B 0,C 180,E1 -2001.913,E2 -2001.913} C_VEL
LIN {X 0,Y 576.713,Z 371.275,A -85,B 0,C 180,E1 -2002.853,E2 -2002.853} C_VEL
LIN {X 0,Y 574.319,Z 371.57,A -85,B 0,C 180,E1 -2003.609,E2 -2003.609} C_VEL
LIN {X 0,Y 573.32,Z 371.697,A -85,B 0,C 180,E1 -2004.193,E2 -2004.193} C_VEL
LIN {X 0,Y 573.254,Z 371.702,A -85,B 0,C 180,E1 -2004.391,E2 -2004.391} C_VEL
LIN {X 0,Y 573.253,Z 371.701,A -85,B 0,C 180,E1 -2006.976,E2 -2006.976} C_VEL
LIN {X 0,Y 573.249,Z 371.704,A -85,B 0,C 180,E1 -2009.488,E2 -2009.488} C_VEL
LIN {X 0,Y 573.256,Z 371.705,A -85,B 0,C 180,E1 -2012.645,E2 -2012.645} C_VEL
LIN {X 0,Y 573.271,Z 371.7,A -85,B 0,C 180,E1 -2015.184,E2 -2015.184} C_VEL
LIN {X 0,Y 573.239,Z 371.704,A -85,B 0,C 180,E1 -2017.807,E2 -2017.807} C_VEL
LIN {X 0,Y 573.272,Z 371.705,A -85,B 0,C 180,E1 -2020.528,E2 -2020.528} C_VEL
LIN {X 0,Y 573.247,Z 371.707,A -85,B 0,C 180,E1 -2023.669,E2 -2023.669} C_VEL
LIN {X 0,Y 573.251,Z 371.703,A -85,B 0,C 180,E1 -2026.642,E2 -2026.642} C_VEL
LIN {X 0,Y 573.262,Z 371.701,A -85,B 0,C 180,E1 -2029.476,E2 -2029.476} C_VEL
LIN {X 0,Y 573.227,Z 371.708,A -85,B 0,C 180,E1 -2031.297,E2 -2031.297} C_VEL
LIN {X 0,Y 573.303,Z 376.47,A -85,B 0,C 180,E1 -2034.006,E2 -2034.006} C_VEL
LIN {X 0,Y 573.288,Z 381.082,A -85,B 0,C 180,E1 -2036.519,E2 -2036.519} C_VEL
LIN {X 0,Y 573.203,Z 386.012,A -85,B 0,C 180,E1 -2039.123,E2 -2039.123} C_VEL
LIN {X 0,Y 573.175,Z 391.548,A -85,B 0,C 180,E1 -2041.986,E2 -2041.986} C_VEL
LIN {X 0,Y 573.118,Z 396.723,A -85,B 0,C 180,E1 -2044.583,E2 -2044.583} C_VEL
LIN {X 0,Y 573.073,Z 403.025,A -85,B 0,C 180,E1 -2047.656,E2 -2047.656} C_VEL
LIN {X 0,Y 573.03,Z 407.752,A -85,B 0,C 180,E1 -2049.915,E2 -2049.915} C_VEL
LIN {X 0,Y 573.045,Z 412.479,A -85,B 0,C 180,E1 -2052.145,E2 -2052.145} C_VEL
LIN {X 0,Y 573.041,Z 418.535,A -85,B 0,C 180,E1 -2054.962,E2 -2054.962} C_VEL
LIN {X 0,Y 574.262,Z 425.044,A -85,B 0,C 180,E1 -2055.108,E2 -2055.108} C_VEL
LIN {X 0,Y 574.128,Z 439.529,A -85,B 0,C 180,E1 -2055.455,E2 -2055.455} C_VEL
LIN {X 0,Y 574.004,Z 453.962,A -85,B 0,C 180,E1 -2055.961,E2 -2055.961} C_VEL
LIN {X 0,Y 573.868,Z 466.52,A -85,B 0,C 180,E1 -2056.545,E2 -2056.545} C_VEL
LIN {X 0,Y 573.683,Z 478.806,A -85,B 0,C 180,E1 -2057.261,E2 -2057.261} C_VEL
LIN {X 0,Y 573.551,Z 491.211,A -85,B 0,C 180,E1 -2058.156,E2 -2058.156} C_VEL
LIN {X 0,Y 573.438,Z 501.707,A -85,B 0,C 180,E1 -2059.081,E2 -2059.081} C_VEL
LIN {X 0,Y 573.245,Z 511.476,A -85,B 0,C 180,E1 -2060.117,E2 -2060.117} C_VEL
LIN {X 0,Y 573.202,Z 519.859,A -85,B 0,C 180,E1 -2061.184,E2 -2061.184} C_VEL
LIN {X 0,Y 573.111,Z 527.87,A -85,B 0,C 180,E1 -2062.425,E2 -2062.425} C_VEL
LIN {X 0,Y 573.022,Z 534.321,A -85,B 0,C 180,E1 -2063.663,E2 -2063.663} C_VEL
LIN {X 0,Y 573,Z 538.798,A -85,B 0,C 180,E1 -2064.722,E2 -2064.722} C_VEL
LIN {X 0,Y 573.029,Z 542.309,A -85,B 0,C 180,E1 -2065.78,E2 -2065.78} C_VEL
LIN {X 0,Y 572.957,Z 545.742,A -85,B 0,C 180,E1 -2067.188,E2 -2067.188} C_VEL
LIN {X 0,Y 572.944,Z 547.783,A -85,B 0,C 180,E1 -2068.594,E2 -2068.594} C_VEL
LIN {X 0,Y 572.937,Z 548.496,A -85,B 0,C 180,E1 -2070,E2 -2070} C_VEL
LIN {X 0,Y 572.942,Z 547.88,A -85,B 0,C 180,E1 -2071.406,E2 -2071.406} C_VEL
LIN {X 0,Y 572.954,Z 545.923,A -85,B 0,C 180,E1 -2072.812,E2 -2072.812} C_VEL
LIN {X 0,Y 573.03,Z 542.578,A -85,B 0,C 180,E1 -2074.22,E2 -2074.22} C_VEL
LIN {X 0,Y 573.056,Z 537.749,A -85,B 0,C 180,E1 -2075.631,E2 -2075.631} C_VEL
LIN {X 0,Y 573.054,Z 531.283,A -85,B 0,C 180,E1 -2077.045,E2 -2077.045} C_VEL
LIN {X 0,Y 573.142,Z 524.083,A -85,B 0,C 180,E1 -2078.284,E2 -2078.284} C_VEL
LIN {X 0,Y 573.218,Z 516.544,A -85,B 0,C 180,E1 -2079.349,E2 -2079.349} C_VEL
LIN {X 0,Y 573.316,Z 507.489,A -85,B 0,C 180,E1 -2080.417,E2 -2080.417} C_VEL
LIN {X 0,Y 573.468,Z 496.53,A -85,B 0,C 180,E1 -2081.487,E2 -2081.487} C_VEL
LIN {X 0,Y 573.606,Z 485.348,A -85,B 0,C 180,E1 -2082.381,E2 -2082.381} C_VEL
LIN {X 0,Y 573.753,Z 472.997,A -85,B 0,C 180,E1 -2083.188,E2 -2083.188} C_VEL
LIN {X 0,Y 573.947,Z 461.114,A -85,B 0,C 180,E1 -2083.815,E2 -2083.815} C_VEL
LIN {X 0,Y 574.094,Z 448.627,A -85,B 0,C 180,E1 -2084.336,E2 -2084.336} C_VEL
LIN {X 0,Y 574.186,Z 435.346,A -85,B 0,C 180,E1 -2084.752,E2 -2084.752} C_VEL
LIN {X 0,Y 574.142,Z 424.018,A -85,B 0,C 180,E1 -2085.006,E2 -2085.006} C_VEL
LIN {X 0,Y 573.037,Z 418.533,A -85,B 0,C 180,E1 -2085.13,E2 -2085.13} C_VEL
LIN {X 0,Y 573.045,Z 412.671,A -85,B 0,C 180,E1 -2087.855,E2 -2087.855} C_VEL
LIN {X 0,Y 573.027,Z 407.941,A -85,B 0,C 180,E1 -2090.085,E2 -2090.085} C_VEL
LIN {X 0,Y 573.074,Z 403.212,A -85,B 0,C 180,E1 -2092.345,E2 -2092.345} C_VEL
LIN {X 0,Y 573.118,Z 396.905,A -85,B 0,C 180,E1 -2095.417,E2 -2095.417} C_VEL
LIN {X 0,Y 573.176,Z 391.736,A -85,B 0,C 180,E1 -2098.014,E2 -2098.014} C_VEL
LIN {X 0,Y 573.204,Z 385.964,A -85,B 0,C 180,E1 -2100.995,E2 -2100.995} C_VEL
LIN {X 0,Y 573.266,Z 381.165,A -85,B 0,C 180,E1 -2103.524,E2 -2103.524} C_VEL
LIN {X 0,Y 573.302,Z 376.539,A -85,B 0,C 180,E1 -2106.045,E2 -2106.045} C_VEL
LIN {X 0,Y 573.226,Z 371.82,A -85,B 0,C 180,E1 -2108.703,E2 -2108.703} C_VEL
LIN {X 0,Y 573.24,Z 371.707,A -85,B 0,C 180,E1 -2111.594,E2 -2111.594} C_VEL
LIN {X 0,Y 573.243,Z 371.705,A -85,B 0,C 180,E1 -2114.333,E2 -2114.333} C_VEL
LIN {X 0,Y 573.243,Z 371.704,A -85,B 0,C 180,E1 -2117.359,E2 -2117.359} C_VEL
LIN {X 0,Y 573.244,Z 371.702,A -85,B 0,C 180,E1 -2120.392,E2 -2120.392} C_VEL
LIN {X 0,Y 573.26,Z 371.702,A -85,B 0,C 180,E1 -2123.078,E2 -2123.078} C_VEL
LIN {X 0,Y 573.276,Z 371.701,A -85,B 0,C 180,E1 -2125.672,E2 -2125.672} C_VEL
LIN {X 0,Y 573.245,Z 371.702,A -85,B 0,C 180,E1 -2128.185,E2 -2128.185} C_VEL
LIN {X 0,Y 573.267,Z 371.703,A -85,B 0,C 180,E1 -2130.634,E2 -2130.634} C_VEL
LIN {X 0,Y 573.255,Z 371.701,A -85,B 0,C 180,E1 -2133.024,E2 -2133.024} C_VEL
LIN {X 0,Y 573.279,Z 371.7,A -85,B 0,C 180,E1 -2135.366,E2 -2135.366} C_VEL
LIN {X 0,Y 573.232,Z 371.704,A -85,B 0,C 180,E1 -2138.419,E2 -2138.419} C_VEL
LIN {X 0,Y 573.273,Z 371.703,A -85,B 0,C 180,E1 -2140.731,E2 -2140.731} C_VEL
LIN {X 0,Y 573.253,Z 371.705,A -85,B 0,C 180,E1 -2143.622,E2 -2143.622} C_VEL
LIN {X 0,Y 573.277,Z 371.7,A -85,B 0,C 180,E1 -2145.807,E2 -2145.807} C_VEL
LIN {X 0,Y 573.267,Z 371.705,A -85,B 0,C 180,E1 -2148.745,E2 -2148.745} C_VEL
LIN {X 0,Y 573.287,Z 371.698,A -85,B 0,C 180,E1 -2151.54,E2 -2151.54} C_VEL
LIN {X 0,Y 573.293,Z 371.696,A -85,B 0,C 180,E1 -2154.372,E2 -2154.372} C_VEL
LIN {X 0,Y 573.307,Z 371.695,A -85,B 0,C 180,E1 -2157.892,E2 -2157.892} C_VEL
LIN {X 0,Y 573.335,Z 371.691,A -85,B 0,C 180,E1 -2160.702,E2 -2160.702} C_VEL
LIN {X 0,Y 573.239,Z 371.706,A -85,B 0,C 180,E1 -2163.514,E2 -2163.514} C_VEL
LIN {X 0,Y 573.291,Z 371.696,A -85,B 0,C 180,E1 -2165.628,E2 -2165.628} C_VEL
LIN {X 0,Y 573.275,Z 371.7,A -85,B 0,C 180,E1 -2167.75,E2 -2167.75} C_VEL
LIN {X 0,Y 573.27,Z 371.698,A -85,B 0,C 180,E1 -2170.597,E2 -2170.597} C_VEL
LIN {X 0,Y 573.269,Z 371.702,A -85,B 0,C 180,E1 -2172.748,E2 -2172.748} C_VEL
LIN {X 0,Y 573.239,Z 371.705,A -85,B 0,C 180,E1 -2174.92,E2 -2174.92} C_VEL
LIN {X 0,Y 573.256,Z 371.707,A -85,B 0,C 180,E1 -2177.848,E2 -2177.848} C_VEL
LIN {X 0,Y 573.255,Z 371.701,A -85,B 0,C 180,E1 -2180.076,E2 -2180.076} C_VEL
LIN {X 0,Y 573.238,Z 371.704,A -85,B 0,C 180,E1 -2183.099,E2 -2183.099} C_VEL
LIN {X 0,Y 573.252,Z 371.702,A -85,B 0,C 180,E1 -2185.41,E2 -2185.41} C_VEL
LIN {X 0,Y 573.255,Z 371.702,A -85,B 0,C 180,E1 -2188.029,E2 -2188.029} C_VEL
LIN {X 0,Y 573.233,Z 371.71,A -85,B 0,C 180,E1 -2190.882,E2 -2190.882} C_VEL
LIN {X 0,Y 573.265,Z 371.7,A -85,B 0,C 180,E1 -2193.524,E2 -2193.524} C_VEL
LIN {X 0,Y 573.264,Z 371.702,A -85,B 0,C 180,E1 -2196.048,E2 -2196.048} C_VEL
LIN {X 0,Y 573.252,Z 371.705,A -85,B 0,C 180,E1 -2198.701,E2 -2198.701} C_VEL
LIN {X 0,Y 573.246,Z 371.703,A -85,B 0,C 180,E1 -2201.594,E2 -2201.594} C_VEL
LIN {X 0,Y 573.227,Z 371.705,A -85,B 0,C 180,E1 -2204.334,E2 -2204.334} C_VEL
LIN {X 0,Y 573.244,Z 371.706,A -85,B 0,C 180,E1 -2207.358,E2 -2207.358} C_VEL
LIN {X 0,Y 573.25,Z 371.708,A -85,B 0,C 180,E1 -2210.393,E2 -2210.393} C_VEL
LIN {X 0,Y 573.259,Z 371.737,A -85,B 0,C 180,E1 -2210.961,E2 -2210.961} C_VEL
LIN {X 0,Y 573.415,Z 374.29,A -85,B 0,C 180,E1 -2212.206,E2 -2212.206} C_VEL
LIN {X 0,Y 573.375,Z 379.869,A -85,B 0,C 180,E1 -2214.824,E2 -2214.824} C_VEL
LIN {X 0,Y 573.294,Z 385.438,A -85,B 0,C 180,E1 -2217.357,E2 -2217.357} C_VEL
LIN {X 0,Y 573.253,Z 391.061,A -85,B 0,C 180,E1 -2219.824,E2 -2219.824} C_VEL
LIN {X 0,Y 573.208,Z 396.677,A -85,B 0,C 180,E1 -2222.231,E2 -2222.231} C_VEL
LIN {X 0,Y 573.176,Z 403.6,A -85,B 0,C 180,E1 -2225.142,E2 -2225.142} C_VEL
LIN {X 0,Y 573.133,Z 409.699,A -85,B 0,C 180,E1 -2227.658,E2 -2227.658} C_VEL
LIN {X 0,Y 573.107,Z 415.27,A -85,B 0,C 180,E1 -2229.918,E2 -2229.918} C_VEL
LIN {X 0,Y 573.085,Z 423.116,A -85,B 0,C 180,E1 -2233.048,E2 -2233.048} C_VEL
LIN {X 0,Y 573.066,Z 427.923,A -85,B 0,C 180,E1 -2234.914,E2 -2234.914} C_VEL
LIN {X 0,Y 574.269,Z 435.02,A -85,B 0,C 180,E1 -2235.062,E2 -2235.062} C_VEL
LIN {X 0,Y 574.143,Z 449.474,A -85,B 0,C 180,E1 -2235.409,E2 -2235.409} C_VEL
LIN {X 0,Y 574.006,Z 463.958,A -85,B 0,C 180,E1 -2235.916,E2 -2235.916} C_VEL
LIN {X 0,Y 573.831,Z 477.388,A -85,B 0,C 180,E1 -2236.544,E2 -2236.544} C_VEL
LIN {X 0,Y 573.682,Z 489.509,A -85,B 0,C 180,E1 -2237.261,E2 -2237.261} C_VEL
LIN {X 0,Y 573.529,Z 500.754,A -85,B 0,C 180,E1 -2238.075,E2 -2238.075} C_VEL
LIN {X 0,Y 573.449,Z 510.847,A -85,B 0,C 180,E1 -2238.955,E2 -2238.955} C_VEL
LIN {X 0,Y 573.269,Z 520.333,A -85,B 0,C 180,E1 -2239.939,E2 -2239.939} C_VEL
LIN {X 0,Y 573.197,Z 528.911,A -85,B 0,C 180,E1 -2241.006,E2 -2241.006} C_VEL
LIN {X 0,Y 573.112,Z 537.115,A -85,B 0,C 180,E1 -2242.248,E2 -2242.248} C_VEL
LIN {X 0,Y 573.036,Z 543.448,A -85,B 0,C 180,E1 -2243.427,E2 -2243.427} C_VEL
LIN {X 0,Y 573.001,Z 548.961,A -85,B 0,C 180,E1 -2244.722,E2 -2244.722} C_VEL
LIN {X 0,Y 573.028,Z 552.442,A -85,B 0,C 180,E1 -2245.78,E2 -2245.78} C_VEL
LIN {X 0,Y 572.956,Z 555.831,A -85,B 0,C 180,E1 -2247.188,E2 -2247.188} C_VEL
LIN {X 0,Y 572.941,Z 557.832,A -85,B 0,C 180,E1 -2248.594,E2 -2248.594} C_VEL
LIN {X 0,Y 572.937,Z 558.5,A -85,B 0,C 180,E1 -2250,E2 -2250} C_VEL
LIN {X 0,Y 572.941,Z 557.833,A -85,B 0,C 180,E1 -2251.406,E2 -2251.406} C_VEL
LIN {X 0,Y 572.956,Z 555.833,A -85,B 0,C 180,E1 -2252.812,E2 -2252.812} C_VEL
LIN {X 0,Y 573.028,Z 552.444,A -85,B 0,C 180,E1 -2254.22,E2 -2254.22} C_VEL
LIN {X 0,Y 573.057,Z 547.568,A -85,B 0,C 180,E1 -2255.63,E2 -2255.63} C_VEL
LIN {X 0,Y 573.065,Z 542.818,A -85,B 0,C 180,E1 -2256.699,E2 -2256.699} C_VEL
LIN {X 0,Y 573.126,Z 536.038,A -85,B 0,C 180,E1 -2257.929,E2 -2257.929} C_VEL
LIN {X 0,Y 573.225,Z 527.559,A -85,B 0,C 180,E1 -2259.171,E2 -2259.171} C_VEL
LIN {X 0,Y 573.304,Z 518.708,A -85,B 0,C 180,E1 -2260.239,E2 -2260.239} C_VEL
LIN {X 0,Y 573.462,Z 507.992,A -85,B 0,C 180,E1 -2261.308,E2 -2261.308} C_VEL
LIN {X 0,Y 573.617,Z 497.144,A -85,B 0,C 180,E1 -2262.201,E2 -2262.201} C_VEL
LIN {X 0,Y 573.733,Z 485.26,A -85,B 0,C 180,E1 -2263.008,E2 -2263.008} C_VEL
LIN {X 0,Y 573.946,Z 472.096,A -85,B 0,C 180,E1 -2263.724,E2 -2263.724} C_VEL
LIN {X 0,Y 574.059,Z 459.049,A -85,B 0,C 180,E1 -2264.277,E2 -2264.277} C_VEL
LIN {X 0,Y 574.221,Z 444.731,A -85,B 0,C 180,E1 -2264.722,E2 -2264.722} C_VEL
LIN {X 0,Y 574.119,Z 433.303,A -85,B 0,C 180,E1 -2264.976,E2 -2264.976} C_VEL
LIN {X 0,Y 573.062,Z 427.806,A -85,B 0,C 180,E1 -2265.106,E2 -2265.106} C_VEL
LIN {X 0,Y 573.088,Z 420.842,A -85,B 0,C 180,E1 -2267.853,E2 -2267.853} C_VEL
LIN {X 0,Y 573.141,Z 413.413,A -85,B 0,C 180,E1 -2270.831,E2 -2270.831} C_VEL
LIN {X 0,Y 573.156,Z 405.985,A -85,B 0,C 180,E1 -2273.869,E2 -2273.869} C_VEL
LIN {X 0,Y 573.193,Z 399.717,A -85,B 0,C 180,E1 -2276.483,E2 -2276.483} C_VEL
LIN {X 0,Y 573.247,Z 392.638,A -85,B 0,C 180,E1 -2279.488,E2 -2279.488} C_VEL
LIN {X 0,Y 573.284,Z 386.359,A -85,B 0,C 180,E1 -2282.233,E2 -2282.233} C_VEL
LIN {X 0,Y 573.367,Z 380.705,A -85,B 0,C 180,E1 -2284.79,E2 -2284.79} C_VEL
LIN {X 0,Y 573.403,Z 375.57,A -85,B 0,C 180,E1 -2287.185,E2 -2287.185} C_VEL
LIN {X 0,Y 573.259,Z 371.736,A -85,B 0,C 180,E1 -2289.039,E2 -2289.039} C_VEL
LIN {X 0,Y 573.255,Z 371.705,A -85,B 0,C 180,E1 -2291.596,E2 -2291.596} C_VEL
LIN {X 0,Y 573.235,Z 371.707,A -85,B 0,C 180,E1 -2294.334,E2 -2294.334} C_VEL
LIN {X 0,Y 573.241,Z 371.704,A -85,B 0,C 180,E1 -2297.359,E2 -2297.359} C_VEL
LIN {X 0,Y 573.25,Z 371.702,A -85,B 0,C 180,E1 -2300.393,E2 -2300.393} C_VEL
LIN {X 0,Y 573.258,Z 371.702,A -85,B 0,C 180,E1 -2303.078,E2 -2303.078} C_VEL
LIN {X 0,Y 573.275,Z 371.702,A -85,B 0,C 180,E1 -2305.672,E2 -2305.672} C_VEL
LIN {X 0,Y 573.243,Z 371.703,A -85,B 0,C 180,E1 -2308.185,E2 -2308.185} C_VEL
LIN {X 0,Y 573.266,Z 371.704,A -85,B 0,C 180,E1 -2310.634,E2 -2310.634} C_VEL
LIN {X 0,Y 573.252,Z 371.701,A -85,B 0,C 180,E1 -2313.024,E2 -2313.024} C_VEL
LIN {X 0,Y 573.277,Z 371.701,A -85,B 0,C 180,E1 -2315.366,E2 -2315.366} C_VEL
LIN {X 0,Y 573.231,Z 371.705,A -85,B 0,C 180,E1 -2318.419,E2 -2318.419} C_VEL
LIN {X 0,Y 573.281,Z 371.702,A -85,B 0,C 180,E1 -2320.728,E2 -2320.728} C_VEL
LIN {X 0,Y 573.251,Z 371.705,A -85,B 0,C 180,E1 -2323.622,E2 -2323.622} C_VEL
LIN {X 0,Y 573.276,Z 371.7,A -85,B 0,C 180,E1 -2325.807,E2 -2325.807} C_VEL
LIN {X 0,Y 573.265,Z 371.704,A -85,B 0,C 180,E1 -2328.745,E2 -2328.745} C_VEL
LIN {X 0,Y 573.286,Z 371.699,A -85,B 0,C 180,E1 -2331.541,E2 -2331.541} C_VEL
LIN {X 0,Y 573.291,Z 371.696,A -85,B 0,C 180,E1 -2334.372,E2 -2334.372} C_VEL
LIN {X 0,Y 573.309,Z 371.695,A -85,B 0,C 180,E1 -2337.892,E2 -2337.892} C_VEL
LIN {X 0,Y 573.333,Z 371.691,A -85,B 0,C 180,E1 -2340.702,E2 -2340.702} C_VEL
